# B&R Automation Studio project NAELD004C00R10L518F00 (part 4)

### Update LogProgram.txt
```
25/9/2023
Solved Inlet Shutter buffer empty close
added interlock to stop traverser and lifter when left or clear sensor sensed

2023-08-21, 2023-09-04, 2023-09-06   (R10)
DInput ,Doutput, OpsLifTrav - added outletshutter 2 (0276)
NtParam,UI - added Trolleylck 1&2 (0258)
UI,mcparam - added lane b fix to fix offset
UI - R to L
2023-09-04
UI - update 0258a topview position, teach picture
OpsMagConvLD1, LD2 - added p_bLinkTrolleyLckPrep
MtrPshr - MtrPshrActRet - added iRetSlwTor
Act_OptP0001Startup - Changed to AND gate.
2023-09-06
p0200 - added manual unlock trolley btn.

2023-07-31 (R9)
DInput - Act_Background - Start up buzzer update
UI - Act_Background - P1000_LangTime - Update the arrangement and display of the languagues and time
Ntparam - Add Chinese & German prep
AutoRcp - update structure , ntparam added eAutoRcpPrecededBy

2023_07_26 continue(R8) General_update
    > Update
            Manual accept for
            1) LFFollower,Follower1,Follower2,etc:Act_Background_AccData
            2) LCSLF:Act_Main
            3) USHermes: Act_Background_AccData

            HMI:
            1) Act_OptP0200ToP0201AccDat(Name based on Project)

2023-07-03 (R8)
-Auto Rcp (Compatiple only with Horizontal Hermes 1.3)
- Magazine auto Calculated width,min,max,pitch based on Board Available and Board Forecast
- Magazine Properties Retain Function
-SvyHermes Board Arrived,Board depart (Slotid,Magazaine ID)
-OPCUA AGV with RFID, read RFID tag when enter, write when exit
-Adding Magazine Exiting with buffer full,release magazine, AGV ready signal , product different (Auto Rcp)
- Error Handling for AutoRcp (Under Testing)
- Tuning MtrPshr
Commission line (_S0)
-MtrPshr - to solve alarm triggered when powered on
-Buffer1,2,3,4 - update Act_Initial diNxtUnloadSlt value.
-OpsTravLifLD - Rls button during readRFID
(_S1)
-Hermes<> smema transition to flush out magazine.
-Debug shutter close when puller extend
(_S2)
-Remove release btn mask.
-Resolved the last board with same width board available. (DSHermes)
(_S3)	2023-07-26
-AutoRcp - Act_Background2 -added p_diRequestedMinSlt when 5mm / 30mm btm clearance
-Debug the right sensor false triggered. (NOT(p_bConvHvBrd)) ,allowed reach ds position without active right sensor
(_S4) 2023-08-11
-Buffer 1,2,3 - Act_Background - added diCurrSltHermes
-DSHermes - seq - boardForcastID - No need sBoardID
			-ProcessData - added timer to reset bSendBFId (Forecast ID)
-SvyHermes - Act_Link - boardArrived - channge to p_bPullerRetRS
-OpsTravLifLD - TravLifLDStep1InletPneuCls - avoid keep open when no curtain sensor
-UI - update product name to WorkOrderId (in Hermes) (done B02,B03)

2023-06-05, 2023-06-14 (R7) --
NtParam - added hermes 1.3 supervisory
		- added shutter2,3 prep
		- added customerReq
AutoRcp - New package.

2023-05-17 (R6) -- .
-Debug the right sensor false triggered. (NOT(p_bConvHvBrd AND p_bRightSen))
OpsTravLifLD -- Added TravLifLDStep1DSSigRechk > TravLifLDStep1ConvEntBrdLostErr
Visu - Show the DBAOnRgt sensor in machine param.
OpsMagConvLD1,2,3 -Added downpulse for clampDetect sensor when magazine pre-exit
P0800, OpsMagConvLD1,2,3 - Updated set magEmpty at magInfo during run.
NtParam - Added eCustomerReq
OpsMagConvLD1 - Act_OpsInfo - Catered 2 empty magazine only buzzer. (BChina)
OpsTravLifLD -- added p_siCntrPullLmt and fbCTDPullLmt

2023-05-08 (R5) --
UI - Act_OptP0400Load.st - Avoid prompt LF message box when error.
OpsTravLifLD - Act_Link - Add a_bRlsMagBtn[1,2,3]
OpsMagConvLD1,2,3 - Act_OpsRun - Added condition on bRlsMagAllw.
HWInfo - Generate MacAddr file.

2023-3-22 (R4) --
Alarm
-Alarm.var added global variable to link text snippet alarm UI
-Act_Background - Recovery list changed to Alarm Error Code
-UI P0200 - change recovery text from string to text group
-UI P0600 - Trigger alarm using bAlm,bWarning,Errcode replacing the original string
-UI P0600 - Adding additional button to check alarm history
-UI Visu  - P0200,P0600 Using given Visu Alarm component instead of string text as the Alarm table

2023-03-15 (R4) --
OpsMagConvLD1,2,3,4 -- added p_bProjLifTravMnlLoad for non roller condition
CPU.sw -- PushPull Cycle time move up to 20 ms same as PullConv

2023-03-03 (R4) --
-UPDATE outstanding:
OpsMagConvLD1,2,3 - Act_OpsRun.st - Make unclamp top clamper when orientation / height sensor fail to sense.
									-LD2 ,3  -Rectified the height sensor alarm when condition not meet.
OpsTravLifLD - Act_OpsSubRun1.st - Catered unclamp(OpsMagConvLD1,2,3) when width check error.
Visu, P0900 , P0201 - Added magazine width check sensor IO.
P0202,P0203,P0204 - Rectified blank IO (Top Rmt Unclamp Sensor)
P1026 ,P1031 - Act_Main, Exit , FBCtrl - Add Bypass curtain sensor on all teaching pages.
DOutput - Act_Link - Allowed UI ctrl in stop mode.
OpsMagConvLD1,2,3 - Act_OpsRun.st - Add fbSelClmpTm wait for penumatic full clamp.
									- Make unclamp fix clamper when orientation / height sensor fail to sense.
PullConv - Local.var - Rearrange the offset text. (puller is Extending/ Retracting)

2023-02-23
LF 	- Act_InitGlobal	- Added p_eProdRcpStat, p_eProdRcpStatus, p_eLinkUIProdRcpAct, p_tyProdRcpCurrRcpWr
	- InputRef_Link		- Added ref variables based on declaration in Act_InitGlobal.
	- Act_Background_AccDat	- Re-adjusted usiProdAccDatStep, and additional usiProdAccDatStep for ProdRcpActWriteCurrRcpParam ProdRcp's Action

**Search Funciton Update** - NtRecipe 5.00.5 (L517)
- ProdRcp - Act_Main & Local.var
- Act_EntP1040Disp
- Act_OptP1040Save
- Act_OptP1040Del
- Act_OptP1040ToXML
- Act_OptP1040FromXML
- Act_EntP0400Disp
2023-01-17 (ANGSY)
UI - Act_Background - Act_OptP1080EditUsr - Add tyStringPw.sValue for every cases of tyP1080UsrMgmt.tyUsrMgmt.tyDrpDnLvl.usiValueIdx
										  - Uncomment tyP1080UsrMgmt.tyEdit.tyStringPw.sValue := '';
- Shift bDBAOnRgtSen from NtParam to McParam
- FTP drive migrate to F drive
--##

2022-12-07 (R3)
Ui - optimization(P0202 ,P0930,P0931, P0932),P0937 -update puller go width
NtParam - Added tyPPTorqParam
Pneu2SenInShutter2 - disabled when single inlet used.
Pneu2SenInShutter3 - disabled when single inlet used.
OpsTravLifLD - OpsRun - added MagPlat_Step1EntBrd, MagPlat_Step1InletPneuCls, MagPlat_Step1InletPneuOpn. (for magazine platform)

2022-09-24,2022-09-25,2022-10-12 (R2)
Trav - Rearrange the alarm list.
OpsTravLifLD - Integrate the individual shutter, cutain sensor feature. -Act_background
			 - Integrate magazine width check
MagConv2Clp1,2,3,4 - Reaccess the Clamping sensor.
PullerPusher - Act_Link - Include interrupt sensor with individual shutter.
			 - Act_RstErr - Reset diJogVel_60FF for recovery.
MagConv2Clp1,2,3 - MagConv2ClpActEntStopClp - changed to Fix clamp then remote clmap.
MagConv2Clp1,2,3 - MagConv2ClpActEntStopClp,MagConv2ClpActEntStopClp - add curtain interrupt for safety clamp
PullConv - Added ConvActInitPuller1 action.
Follower2 - Act_Link - Added p_bAccNewRcpCond.

2022-09-15 (R1)
Buffer 1;2;3;4 - Act_Main - BufferActUnload -make Slt to Slt as positive
Physical view - FTP server - added user for FTP access ProductRecipeXml

2022-03-24 (NAELD004-R0)
Act_Main_P0200 - added RS232Prep and WorkOrder string on barcodeScan
Act_OptP0200BarCodeChgRcp - added bWorkOrderDisp.
Added Act_OptP0200WorkOrderToLMC.st
PullConv - Hold postition when Antijam activated.

2022-03-14
ProdRcp - Act_Main, Local.var
MagRcp - Act_Main, Local.var

2022-02-17
LFFollower, Follower1 - Act_Background - Add p_bDBAOnWOAllign to fbFolllower to send DBA even width check sensor is not alligned.
CANOpenServo - Act_Background - Add error code for Estun Servo Motor.
				              - Reset control word 6040.4 to 0 when servo motor is in position

2021-09-30
Hermes Program - Update
USHermes Program - Update
DSHermes Program - Update
RmtHermes Program - Update
SvyHermes Program - *NEW*
NtParam  - Add new variables for Hermes v1.3
McParam  - Update
Alarm - Update
Startup - Update
UI HMI & Program P0201 - Update
UI HMI & Program P1021 - Update
UI HMI & Program P1022 - Update
UI HMI & Program P1023 - Update

2021-09-02
Revision - R15 , L512
- Width Offset move to NtParam
- Add BadBrdRedLight in NtParam and P0200 for 2021-0532G.
- McMode2 for 2021-0532G in P0201,P0400,P1021,P1040
LFLeader, LFFollower - Local,Input_Ref variables - Modify Product Recipe Related Variables to STRING[254]
LFFollower - Act_Background - Modify bUSAllow To Include p_bInternalReqProdRcpDiff

2021-08-31
Revision - R14 , L512
LFFollower - Update Act_Background
Follower1 - Update Act_Background
- Update NtUSB to 5.00.5
- Update NtLF to 5.01.4
- OPC-UA Security Policy Basic256 Sha256 prohibited

2021-08-02
USB scanner function added.
AIV OPCUA, Hardwired IO and Disabled function added.
IO assignment at physical view changes without alter the value of digital input and digital output at NtParam.

2021-04-06
UI - Visu - Update for 254 Prod Rcp Pop Up
UI - Act_Background - ADD Act_OptP0400RcpPopUp.st & Act_OptP1040RcpPopUp.st & Update Act_OptP0400Preview.st for 254 Prod Rcp Pop Up

2021-02-24
LFLeader - Act_Main - add input to select sequential mode (one time or always active)

2021-02-17
CANOpenServo - Act_Background - PosDiff updated from 50 to 500.
			 - Act_Alarm - udiCode change to 10299
			 - Local.var - update alarm message a_tyAlmText[10298] and a_tyAlmText[10299]

2020-12-14
Update in Act_ChgPage & Act_OptP00001Startup

2020-11-11
Tuning.diAsdaA2FirstTorqueCmd default setting is 300 in NtParam for all Delta servo motor.

2020-10-05
Startup - Act_Main_GetHWInfo - Debug Steps In Network Recovering
LFLeader - Act_Initial, Act_Background_Process and Local.var - Rename and change the type of fbBlkUS to fbBlkUSDS
LFFollower, Follower1 - Act_Background, Act_Background_AccData - Add bLeaderOnline replacing the direct usage of tyLeaderInfo.bOnline
TLBuz - Add Buzzer For All Act_Backgrounds Change Manual Mode Towerlight To Cater For Error Indication
HWInfo - Act_Main - Add IF-ELSE Statement For Simulation, Update Alarm Code for fbGetETHConfigMode & fbSetETHConfigMode
		 Local.var - Add New Alarm Code fbGetETHConfigMode & fbSetETHConfigMode

2020-09-22
LFFollower - Reset bLeaderSeqCtrlInActive in Act_Main_Disable.
HWInfo.typ - Add One Enumeration (eNetworkConfigMod) & Two Actions (fbGetETHConfigMode and fbSetETHConfigMode) - Retrieve Or Set Network Configuration Of The PLC.
HWInfo Init, InitGlobal, InitLocal, Act Main, Act_Initial, Local.var and InputRef.var - Add The Additional Actions Related Variables
McParam  - McParam.typ Add eNetworkMod in tyMcParam.
NtParam  - NtParam.typ Add tyNetworkMOde (UILmt) in tyNtParam.
Startup	   - InitGlobal, InitLocal, Act_Main_GetHWInfo - Add Function To Load Saved Network Configuration s When New Configuration Detected.
		   InputRef_Link.var, InputRef.var & Local.var - Add New Startup Function Variables.

2020-09-16
McParam  - McParam.typ Add sIPAddr & sSubnetMask in tyMcParam.
Startup	 - Init, InitGlobal, InitLocal, Act_Main_GetHWInfo - Add Function To Load Saved IP Parameters When New IP Detected.
		   InputRef_Link.var, InputRef.var & Local.var - Add New HWInfo Function Variables.

2020-09-10
USHermes - Init, Cyclic, Act_Background_TCPConnect, Act_Alarm5 - Improvise Alarm For Connection Lost.
		   Local.var - Add New Alarm Variables & Modify Alarm Text.
DSHermes - Init, Cyclic, Act_Background_TCPListen, Act_Alarm4 - Improvise Alarm For Connection Lost.
		   Local.var - Add New Alarm Variables & Modify Alarm Text.

2020-08-17
LibVer - Act_Main - Modify Function To Function Block In LibVerActReadChk.
		 Act_Initial - Initialize Newly Added Function Blocks.
		 Local.var - Declare New Function Blocks.

2020-08-06
NtParam.typ - Add Two Actions (NtParamSave and NtParamLoad) - Export and import NtParam in XML Format
NtParam Act Main, Act_Initial, tyNtParam, InitLocal, Local.var and InputRef.var - Add The Additional Actions Related Variables
TLBuz - All Act_Backgrounds Change Manual Mode Towerlight To Cater For Error Indication
LFLeader - Add More Tags For Improving Leader Follower Concept, Modify p_diReqProdWidth To Use Downstream Width
LFFollower, Follower 1 	- Add fbOnlineChk For Leader Online Status
						- Modify Act_Initial,Act_Background, Act_Background_AccData
						- Add eCurrMachineStat For Status Indication
ProdRcp.typ		- Add second width
LibVer - Act_Main - Modify LibVerActReadChk, Add Step To Check File Validity.
		 Local.var - Add Alarm Text For File Coruption.

2020-07-24
MagRcp -  Add One Action in Act Main - MagRcpActSort
ProdRcp, MagRcp - p_sSearch and sSearch in Local changed to STRING[254]
ProdRcp, MagRcp - sRcpNm for RcpParam in both ProdRcp.typ and MagRcp.typ temporary changed to STRING[30]

2020-06-30
Revert Traverser Main.st and AWClose Background.st program.
Add Estun error code "65362: sAxisErrTxt := 'Torque output alarm'";

2020-06-08
ProdRcp - Increase Product Recipe Name Length to 254, Add Two Actions in Act Main - ProdRcpActSort & ProdRcpActEndCharFilter
LibVer - Act_Main - LibVerActReadChk, made error if library data files corrupted.

2020-06-05
MagConv - Update the Status of Mag Conv.Add one Action - MagConvActEntToMid.

2020-06-01
Stepper - New package for stepper control.
MotorBrk - Renewed package. Added MotorBrkActSetMtrDirOrCCW1 and MotorBrkActRstMtrDirOrCCW1.
	 	 - Modified fbRotCW and fbRotCCW and the access type to fbConvSenToSenBrkTm2Lmt.
	 	 - Added diMtrSigOnDlyTm (500), diMtrDirOffDlyTm (500), diMtrBrkOnDlyTm(100).

2020-04-28
MagConv - Add MagConvActEntToMid Action.

2020-03-20
NtParam  - Add the selection of Motor model.

2020-03-16
TLBuz - Add two inputs for buzzer behaviour, towerlight flash function to act_background and reset fbwarning.

2019-12-24
LFLeader - Remove fbBlkDS2 in Act_Initial & Act_Background_Process, add pa_bLFOnline in Act_Background_Process

2019-10-31
TLBuz - Regroup Structure Into Nutek, Aptiv & MEK.
MagConv - Separate Program Into MagConv1Clamper & MagConv2Clamper.

2019-10-21
MagConv - Improve with Action MagConvActPreExit & MagConvActPreExitClpr.
LFFollower - Improve Change All Function Without Manually Accept Data.
LFLeader - Add Second Oven Index, Improve Change All Function Without Manually Accept Data.
OpcUaMap.uad - Enable bBypassMnlAccDat Tag Name.
Startup - Act_Main_SDOWrite, Remove SDOWrite.
CANOpenServo - Change Structure Of SDOWrite And Abnormal Movement.

2019-07-30
CANOpenServo - Due To Upgrade of NtMotion.

2019-07-18
LFFollower - Act_Link, Minor debug.

2019-07-15
LCS - Act_Link, Check Recipe Name Must Not Exceed 15 Char.

2019-07-10
LCS - Add More Parameter For Live Data.

2019-07-04
LFFollower - Improve of Recipe Compare Method For p_tyInternalReqProdRcp, tyUpdtProdRcp & tyRlsBrdProdRcpNm.

2019-07-03
LFFollower - Improve Act_Background To Check Whole Product Recipe Different Instead of Name & Width Only.
Buffer - Add p_tyBufferStat & p_tyDispBuffer And Improve For Two Program Control One Memory.

2019-06-28
USHermes - Improve of Act_Background_AccData.
DSHermes - Move of Act_Background_ChgConfig.
Buffer - Improve of bParamDiff Condition.
LCSLF - Improve of LCSActRunProd.

2019-06-27
LFFollower - Improvement To Change Name & Width To Whole Product Recipe Type.

2019-06-17
Conv - Add Two Action : ConvActEntToInOff & ConvActRevImmedStart.

2019-06-12
LFFollower - Add Act_Background_ChkRlsBrd. Improvement of Act_Background_UpdtData.
LCSLF - Add Update Data in Act_Background.

2019-06-11
TLBuz - Modify ChgRcp.
LFFollower - Improvement of UpdtData.

2019-06-10
ProdRcp - Update tyCurrRcp To a_tyCurrRcp (Array).
LFFollower - Add p_bInternalUse.
USHermes - Add p_bInternalUse.
DSHermes - Add p_bInternalUse.

2019-06-07
TLBuz - Add Warning & ChgRcp.
TCP - Add Start Code & End Code Checking.
Buffer - Improve bParamDiff. Add bFIFOOld.

2019-06-04
USHermes - Improvement At Accept Date (Act_Background_AccData).

2019-06-02
TCP - New.

2019-05-30
Hermes - Debug CheckAlive. SequenceTO Start Only After Connection Establish.
Flatstream - Debug Act_Main.
USHermes - Update Act_Link to Accept New Recipe.

2019-05-29
DVFrame - Change From RS232. Improvement & Debug.
Flatstream - New.

2019-05-28
MagConv - Add MagConvActInitClpStop.
DCConv - Improvement of DC Motor Alarm Trigger Time.
LFFollower - Improve of Act_Background.
LCS - Add "Warning" & "Info" For Live Data.

2019-05-27
LFFollower - Debug Act_Link.
LCS - Debug Act_Link. Add sErrMsg.
Buffer - Debug Act_Main_Bffr. Add bMagRemoved.
Data - Update of Default User.dat.

2019-05-24
LFFollower - Improve of Act_Background.
MagConv - Add MagConvActEntClpStop.
TLBuz - Modify Warning Condition.

2019-05-22
OpcUaMap.uad - Update Tag Name.
LF - Modify Set Time. Improve Of Act_Background for Accept Data.
LFLeader - Add New Tag Name.
Time - Update of Act_InitGlobal For LF Sync Time.
LCS - Update To Reset If Receive Idle From LCS.

2019-05-21
RS232 - Add FullReadUntilValid.
LCS - Move Some Program From Act_Background To Act_Link. Bug Fixed.

2019-05-20
RS232 - Modify to work with start code & end code.
ProdRcp - Modify on dtLastModified in Act_LinkAction.
LCS - Act_Background Show Boolean & dtLastModified Working Sample. Add Function Enable.
TLBuz - Add Aptiv Mode.

2019-05-18
Buffer - Check Next Unload Ignore Product Name.

2019-05-15
OvenInfo - Improve of Act_Background.
Buffer - Add bParamDiff to check current parameter and request parameter different.

2019-05-14
LCS - Update Act_InitGlobal.
RS232 - New.

2019-05-11
LFFollower - Improve And Able To Ignore MagRcp If Necessary.

2019-05-10
TLBuz - Add Simulation Mode.
ProdRcp - Improve Act_LinkAction.
Buffer - Improve Act_LinkAction.
HWInfo - Improve Act_Main While In Simulation.

2019-05-09
CANOpenServo - Improve of Error Axis Move Abnormally By External Force (10000).
ProdRcp - Debug Write Recipe. Add Save List.
MagRcp - Debug Write Recipe. Add Save List.
UsrFolder - Create LCS Directory.
Startup - Act_Main_UsrFolder, Create LCS Directory.
Alarm - Combine Two Alarm Info.

2019-05-08
RmtHermes - Debug Log title.
UsrMgmt - Add Access Right Output.

2019-05-07
MagConv - Debug.
ConvBffr - Add Individual Have Board Output.
LF - Major update.
LCSLF - Change Name to tyCurrProdRcp.
ProdRcp - Add Write Recipe Parameter.
MagRcp - Add Write Recipe Parameter.
LCS - Update to match LCS (PC).

2019-05-04
MagRcp - Split Current Magazine Recipe From McParam.
ProdRcp - Split Current Product Recipe From McParam.
UsrMgmt - Split Access Right From McParam. Remove Nutek User.
Hermes - Split Configuration From McParam. Add RmtHermes.
Startup - Split Parameters From McParam. Add RmtHermes.
Remove "File Device" "NutekUser". Please Refer Configuration "4PPC30_043F_21F001".

2019-05-01
Hermes - Log file change to day instead of hour. Due to startup too long to check old log when production run for long.

2019-04-30
LCS - Improve To Match LCS (PC).
LFLeader - Make a_tyFollowerToLeaderTag as Output.
All - sStatTxt & a_sStatText Change To String[200].
ProdRcp - Modify For LCS.

2019-04-28
MpProdRcp - New.
Add "Config.mprecipexml" Under Configuration View > mapp. Please Refer Configuration "4PPC30_043F_21F001".
Add "File devices" For "MpProdRcp". Please Refer Configuration "4PPC30_043F_21F001".
Startup - Modify Due To MpProdRcp.

2019-04-27
DSSMEMA - Update due to NtSMEMA upgrade.

2019-04-26
Buffer - Debug tyBuffer to p_tyBuffer. Improve bLastProductUnload Condition In Unload Board.
Startup - Get Retain ConvBffr.
ConvBffr - Update Link with Startup. Improve bLastProduct Condition In Remove Board. Add Have Board Output.
LFFollower - Improve Act_LinkEn. Add Condition in Act_Link to update current recipe into leader tag.

2019-04-25
LibVer - Modify To Move LibVer From "Private" To "User".
Update "File devices" For "LibVer". Please Refer Configuration "4PPC30_043F_21F001".
Add "File devices" For "LCS". Please Refer Configuration "4PPC30_043F_21F001".
Modify "FTP Server" "Users". Please Refer Configuration "4PPC30_043F_21F001".
Modify "OpcUaMap.uad". Please Refer Configuration "4PPC30_043F_21F001".
LFLeader - Improvement.

2019-04-24
CANOpenServo - Add actual limit sensor output.
ProdRcp - Add "Add" & "Edit" action. Improve of Act_LinkAction to suit LCS.
LCS - New.

2019-04-23
LFLeader - New.

2019-04-21
USHermes - Modify Alarm Info.
LFFollower - New.

2019-04-18
ConvBffr - New.
Buffer - Change of NtBffr.

2019-04-17
CANOpenServo - Remove Extra Homing Parameter, All Use Under tyMotionCANParamInHm.

2019-04-16
Operations - Remove Accept Data & New Data.
Hermes - Debug Log File. Modify Accept Data.

2019-04-11
USHermes - Debug Log by adding step. Add p_bAccDataRdy.
DSHermes - Debug Log by adding step.

2019-04-10
Startup - bNtSettingsLoadDone should be FALSE as default.

2019-04-09
Ops2 - Update of p_bAccDat interlock by Ops1.
USHermes - Update AccDatStep in Act_Link. Remove p_bChkBrdAvl. eStatus2 = Error then bRdyRcv = false. Update Act_Background_BoardAvailableChk. Add Manual Accept Data.
DSHermes - Make local.var BoardAvailable new board parameter to default value.
NtParam - Change of Act_LinkAction.
TLBuz - Change of Act_LinkAction.
Buffer - Change of Act_LinkAction.
Conv - Change of Act_LinkAction.
DCConv - Change of Act_LinkAction.
MagConv - Change of Act_LinkAction.
MotorBrk - Change of Act_LinkAction.
ConvSpd - Change of Act_LinkAction.
SMEMA - Change of Act_LinkAction.
Pneu - Change of Act_LinkAction.
CANOpenServo - Change of Act_LinkAction.
Hermes - Change of Act_LinkAction.

2019-04-08
DSHermes - Minor debug on fbParseBrdAvlExternal.
Hermes - Add program Hermes for board available memory use.
Startup - Due to change of Hermes.

2019-04-04
OvenInfo - Add p_bBGRun.
Startup - Change eStartupStep member order for better display in UI.
UsrMgmt - Add UsrMgmtActUsrBypassLogin & UsrMgmtActNtBypassLogin.
DSHermes - Debug BoardAvailable for "New" and "External".
UI - Remove Not Use Page.

2019-03-29
All - Add Act_LinkAction.

2019-03-28
Startup - Change "DelOldLogFile" to "Alarm". Add "Hermes". Error will reset Action to IDLE.

2019-03-25
All - Change Action become input. Merge Alarm Text & Recovery Text into one type.

2019-03-22
Startup - Add bNtSettingsLoadDone. Move StartupStepParameter after StartupStepUsrFolder in Act_Main.st.
All - Update to match latest method of NtParam.

2019-03-16
Startup - Act_Main_Bffr. Add BufferActBGStartCoolFan in Step 8.

2019-03-15
Hermes - New Release

2019-03-13
UsrFolder - Debug of Log directory path. Add "FileDevice" for "Log".

2019-03-11
DCConv - Minor debug.

2019-02-26
AWClose - Minor debug.

2019-02-23
Alarm - Minor debug.
UsrFolder - Add Create Log Directory.
Startup - Improve of "Act_Main_UsrFolder" due to UsrFolder update.

2019-02-22
CANOpenServo - Change of Act_Action.

2019-02-21
DOutput - Add Act_Link.

2019-02-20
DCConv - Debug of ConvEngage.
CANOpenServo - fbModuleOK delay time change to 5s.

2019-02-19
CANOpenServo - Reset Error need to reset control word 6040.
TLBuz - Improve of condition while p_bManual = True.

2019-02-18
Buffer - Add background control of cool fan run.

2019-02-15
Conv - Improve of condition while p_bManual = True.
DCConv - Improve of condition while p_bManual = True.
MagConv - Improve of condition while p_bManual = True.
MotorBrk - Improve of condition while p_bManual = True.
SMEMA - Improve of condition while p_bManual = True.

2019-02-14
ConvSpd - Improve of condition while p_bManual = TRUE.
Change of Cyclic Time.
CANOpenServo - Change of Position Different Threshold.
Convert Library Into Binary

2019-02-11
TLBuz - Warning Rest Time Change To 5s.
Buffer - Add Magazine Present Timer.

2019-01-27
Buffer - Add error code.

2019-01-26
Buffer - Debug.

2019-01-25
Buffer - Debug a_bSkip array size.
Lifter - Debug Act_Background.
User.dat & NtUser.dat update.

2019-01-24
Pneu - Modify Cyclic for disable.
AW - Add GoWidthOff to turn off motor after auto width move.
Lifter - Debug.
Traverser - Debug.
Buffer - Debug. Add background update display.
OvenInfo - Modify Act_Main_Disable.

2019-01-23
Lifter - Major debug in slot calculation. Add FullMovRel.
CANOpenServo - Debug reset error. Debug Act_Alarm.
DCConv - Debug reset error.
Machine - Debug reset error.
Operation - Debug reset error.

2019-01-22
CANOpenServo - Minor debug.

2019-01-21
DInput - Debug reset error.
CANOpenServo - Add eMainStatus. Add bJogging.
Time - Add eMainStatus.
Operations - Rename eStatus & udiStatus.

2019-01-20
Operations - Update Structure.
SMEMA - Update due to Library update.
Buffer - Add error code.

2019-01-19
TLBuz - Add Warning.

2019-01-18
RstErr - Act_Main update.
CANOpenServo - Add output. Set Default Value for siModOfOptDisp_6061:=6.
Change of Cyclic time.
Buffer - Update Local.var
Add file for NtUser, LibrariesVersion & User.
Conv - Add Pneu status output.
DCConv - Add Pneu status output.
Operations - Modify structure in Cyclic.

2019-01-17
DCConv - Act_Main debug.

2019-01-16
Trav - Remove diPitch.
Lifter - Remove diPitch.
Operations - Modify Reset methos.

2019-01-15
McParam - File name as input.
NtParam - File name as input.
Buffer - File name as input.
Operations - Add bAccData.

2019-01-14
Operations - Update Alarm & Sequence.
SMEMA - bTimer & bVirtual as output. Debug Act_Background timer interlock.

2019-01-12
Conv - Convert time out type.
DCConv - Convert time out type.
MagConv - Convert time out type.
OvenInfo - diBrdInOven change to retain.
SMEMA - Update timer condition. Add bComplSigOn.
Startup - Debug for HWInfo.

2019-01-11
SMEMA - Minor debug. Add Act_LinkEn.
Operations - Add alarm. Add Act_LinkEn.
MagRcp - Add Act_LinkEn.
OvenInfo - Add Act_LinkEn. Minor debug.
Conv - Add Act_LinkEn. Add conveyor time out.
DCConv - Add Act_LinkEn. Add conveyor time out.
MagConv - Add Act_LinkEn. Add conveyor time out.
MotorBrk - Add Act_LinkEn.
ConvSpd - Add Act_LinkEn.
RS232Mirtec - Add Act_LinkEn.
Pneu - Add Act_LinkEn.
CANOpenServo - Add Act_LinkEn. Major Update.

2019-01-10
McParam - Remove ProdRcpWrite & MagRcpWrite.
OvenInfo - Act_Main modify for change of eStat.
Conv - Act_Main modify for change of eStat.
DCConv - Act_Main modify for change of eStat.
MagConv - Act_Main modify for change of eStat.
MotorBrk - Act_Main modify for change of eStat.
ConvSpd - Act_Main modify for change of eStat.
SMEMA - Act_Main modify for change of eStat.
DOutput - Act_Main modify for change of eStat.
Pneu - Act_Main modify for change of eStat.
Operations - Act_Main modify for change of eStat.

2019-01-09
AW - Update bWidthPosDiff when disable.
Lifter - Update bSltPosDiff when disable.
Conv - Add bGdBrdInit. Debug tMtrOffDlyTm. Improve Act_Action to let eStatus = DONE also able change eStat directly.
DCConv - Add bGdBrdInit. Improve Act_Action to let eStatus = DONE also able change eStat directly.
SMEMA - Add tRstDlyTm. Improve Act_Action to let eStatus = DONE also able change eStat directly.
Operations - Add Act_Main_Disable. Improve Act_Action to let eStatus = DONE also able change eStat directly.
TLBuz - Improve Act_Action to let eStatus = DONE also able change eStat directly.
OvenInfo - Improve Act_Action to let eStatus = DONE also able change eStat directly.
MagConv - Improve Act_Action to let eStatus = DONE also able change eStat directly.
MotorBrk - Improve Act_Action to let eStatus = DONE also able change eStat directly.
ConvSpd - Improve Act_Action to let eStatus = DONE also able change eStat directly.
DOutput - Improve Act_Action to let eStatus = DONE also able change eStat directly.
Pneu - Improve Act_Action to let eStatus = DONE also able change eStat directly.

2019-01-08 //Until Here////
DOutput - Add output.
SMEMA - bTimer will be trigger only during SMEMAActRun.
Operations - Combine Ops1 & Ops2 into Ops.

2019-01-07
SMEMA - Add bUSRdy, bUSGdBrdRdy & bDSRdy for USSMEMA & DSSMEMA.
Conv - Add tMtrOffDlyTm.
DCConv - Add tMtrOffDlyTm.
MagConv - Add tMtrOffDlyTm.
Time - Combine Error
CANOpenServo - Combine Error
Alarm - Remove link data.

2019-01-04
Machine - Debug Act_Alarm1.
Time - Debug Init.st.
Operations - Debug Ops1 > Act_Main. Add sStepTxt into Act_Main. Add Act_Dummy.
Conv - Due to NtConv update, add one more type of Exit.
DCConv - Due to NtConv update, add one more type of Exit.
MagConv - Due to NtConv update, add one more type of Exit.
SMEMA - Add Timer & Virtual.

2019-01-03
Machine - Debug Act_Alarm & Act_Alarm1. Modify background error handling.
CANOpenServo - Modify background error handling. Update sStatTxt in Act_Initial.
AW - Replace diStandPitchInUM (Input) to diPitchInUM (Local).
Time - Modify background error handling. Update sStatTxt in Act_Initial.
DCConv - Modify background error handling. Update sStatTxt in Act_Initial.
DInput - Modify background error handling.
UsrMgmt - Update sStatTxt in Act_Initial.
McParam - Update sStatTxt in Act_Initial.
NtParam - Update sStatTxt in Act_Initial.
ProdRcp - Update sStatTxt in Act_Initial.
MagRcp - Update sStatTxt in Act_Initial.
HWInfo - Update sStatTxt in Act_Initial.
UsrFolder - Update sStatTxt in Act_Initial.
LibVer - Update sStatTxt in Act_Initial.
General - Update sStatTxt in Act_Initial.
TLBuz - Update sStatTxt in Act_Initial.
OvenInfo - Update sStatTxt in Act_Initial.
Buffer - Update sStatTxt in Act_Initial.
RstErr - Update sStatTxt in Act_Initial.
Conv - Update sStatTxt in Act_Initial.
MagConv - Update sStatTxt in Act_Initial.
MotorBrk - Update sStatTxt in Act_Initial.
ConvSpd - Update sStatTxt in Act_Initial.
Alarm - Update sStatTxt in Act_Initial.
RS232Mirtec - Update sStatTxt in Act_Initial.
SMEMA - Update sStatTxt in Act_Initial.
UI - Update sStatTxt in Act_Initial.
DOutput - Update sStatTxt in Act_Initial.
Pneu - Update sStatTxt in Act_Initial.
Operations - Update sStatTxt in Act_Initial.
Startup - Update sStatTxt in Act_Initial.

2019-01-02
UsrMgmt - Change of sStatTxt update.
McParam - Change of sStatTxt update.
NtParam - Change of sStatTxt update.
ProdRcp - Change of sStatTxt update.
MagRcp - Change of sStatTxt update.
Time - Change of sStatTxt update.
HWInfo - Change of sStatTxt update.
UsrFolder - Change of sStatTxt update.
LibVer - Change of sStatTxt update.
General - Change of sStatTxt update.
TLBuz - Change of sStatTxt update.
OvenInfo - Change of sStatTxt update.
Buffer - Change of sStatTxt update.
RstErr - Change of sStatTxt update.
Conv - Change of sStatTxt update.
DCConv - Change of sStatTxt update.
MagConv - Change of sStatTxt update.
MotorBrk - Change of sStatTxt update.
ConvSpd - Change of sStatTxt update.
Alarm - Change of sStatTxt update.
RS232Mirtec - Change of sStatTxt update.
SMEMA - Change of sStatTxt update.
UI - Change of sStatTxt update.
DOutput - Change of sStatTxt update.
Pneu - Change of sStatTxt update.
Operations - Change of sStatTxt update.
CANOpenServo - Change of sStatTxt update. Update eStatus to Busy while running.
Startup - Change of sStatTxt update.

2018-12-31
CANOpenServo - Seperate input reference.

2018-12-27
Time - Remove bBGRun.
TLBuz - Remove bBGRun. Add manual reset.
OvenInfo - Background direct link to input bPrepExtdd, bEnExtdd & bDisExtdd. Add manual reset.
Buffer - Background Cool Fan Control direct link to input bPrepCoolTm & bCoolFanTm.
DCConv - Remove bBGRun. Add manual reset.
AlarmLog - Background run is control by Action.
Machine - Remove bBGRun.
SMEMA - Remove bBGRun. Add manual reset.
DInput - Remove bBGRun.
DOutput - Remove bBGRun. Add manual reset.
CANOpenServo - Remove bBGRun. Background run is control by Action. Add manual reset.
AW - Add bWidthPosDiff.
Lifter - Add bSltPosDiff.
Startup - Background run is control by Action. Shorten local variable name.
McParam - Add McParam program without Magazine (McParam2).
RstErr - Add manual reset.
Conv - Add manual reset.
MagConv - Add manual reset.
MotorBrk - Add manual reset.
ConvSpd - Add manual reset.
Pneu - Add manual reset.

2018-12-26
CPU - Update distribute of program in CPU. Update cyclic time.
FTP - Update of FTP server configurations.
Startup - Remove bStartupErr.
HWInfo - After set new IPAddr & Subnetmask will update output.
TLBuz - Rising of bManual will set Amber Light ON.
Conv - Remove functions reset in individual eStat.
MagConv - Remove functions reset in individual eStat.
MotorBrk - Remove functions reset in individual eStat.
DCConv - New program.
Operations - Update of OperationsActStep.

2018-12-24
Operations - Add bRun.Sequence will execute base on bRun instead of bStatusRun.

2018-12-21
Buffer - Add individual cooling fan control.
McParam - Move Hermes parameter to Hermes program type.
MagConv - Add bClprTwoOutputControl. Remove bClprUnclampCtrl.

2018-12-20
TLBuz - Add bMuteBuz.
OvenInfo - Add bDis.
Conv - Add bEn.
MagConv - Add bEn.
MotorBrk - Add bEn.
ConvSpd - Add bEn.
RS232Mirtec - Add bEn.
SMEMA - Add bDis.
Pneu - Add bEn.
CANOpenServo - Add bEn.
CANOpenServo - AutoWidth - Add diMaxWidthInUM, diMinWidthInUM, diWidthOffsetInUM & diStdPitch.
Operations - Add bPrep, bEn & bDis. Add OperationsStatusCycleStopping. Default Status is OperationsStatusStop. Add Boolean output for Status.
MagRcp - Change sDisplayInfo & Magazine Parameter.
Startup - Add bRun.

2018-12-14
RstErr - Add bManual to control reset of output in Idle. Reset output in Idle after ManualMode off.
Conv - Add bManual to control reset of output in Idle. Rename eAction. Reset output in Idle after ManualMode off.
ConvSpd - Add bManual to control reset of output in Idle. Reset output in Idle after ManualMode off.
MtrBrk - Add bManual to control reset of output in Idle. Rename eAction. Reset output in Idle after ManualMode off. Reset after change eStat.
MagConv - Add bManual to control reset of output in Idle. Rename eAction. Reset output in Idle after ManualMode off. Reset after change eStat.
OvenInfo - Set bOvenAllow to TRUE, if all functions not activated.
SMEMA - Reset output in Idle after ManualMode off.
Pneu - Add Extended & Retracted output.

2018-12-13
Conv - Change of Conv2Sen to Conv. Add Reject & Inspection functions. Add individual output control.
Pneu - Add bTwoCtrlIn & bTwoCtrlOut.
TLBuz - Add individual output control.
ConvSpd - Add individual output control.
OvenInfo - Add individual output control. Move functions into Act_Background.
RstErr - Add individual output control.
MtrBrk - Add individual output control.
MagConv - Add individual output control.
DOutput - Add individual output control.
SMEMA - Add individual output control.

2018-12-12
Startup - Add Logout during User Management Startup.
Time - Move Act_Background above Act_Main.
Buffer - Move Act_Background above Act_Main.
Alarm - Move Act_Background above Act_Main.
CANOpenServo - Move Act_Background above Act_Main.
Operations - Change of Conv2Sen to Conv.

2018-12-11
DOutput - Split to Act_InitGlobal & Act_InitLocal.
Pneu - Change in all program. Add Pneu3Sen program.
Operations - Update sample to 2 operations. Rename variable.
CANOpenServo - Rename variable.
```

- LibrariesVersion.dat (binary file, 2222 bytes)
### SoftwareVersion.var
```iecst
VAR CONSTANT
	sSWVersion : STRING[30] := 'NAELD004C00R10L518F00'; (*LifterPlatform and TraverseLifting*)
END_VAR
```

- Visualisation Logical/UI/Visu (not shown)

### UI.typ - Do Not Change!!!
```iecst
(*2019-03-25*)
(**)

TYPE
	eUIAction :
		(
		UIActIdle,
		UIActInitial
		);
END_TYPE

(**)
(*Data*)

TYPE
	eUIInitial :
		(
		UIInitialC0005,
		UIInitialC0007,
		UIInitialP0000,
		UIInitialP0002,
		UIInitialP0200,
		UIInitialP0201,
		UIInitialP0202,
		UIInitialP0203,
		UIInitialP0204,
		UIInitialP0205,
		UIInitialP0206,
		UIInitialP0300,
		UIInitialP0400,
		UIInitialP0410,
		UIInitialP0800,
		UIInitialP0900,
		UIInitialP0910,
		UIInitialP0920,
		UIInitialP0921,
		UIInitialP0923,
		UIInitialP0930,
		UIInitialP0931,
		UIInitialP0932,
		UIInitialP0933,
		UIInitialP0934,
		UIInitialP0935,
		UIInitialP0936,
		UIInitialP0937,
		UIInitialP0939,
		UIInitialP0940,
		UIInitialP0950,
		UIInitialP1000,
		UIInitialP1020,
		UIInitialP1021,
		UIInitialP1022,
		UIInitialP1023,
		UIInitialP1024,
		UIInitialP1025,
		UIInitialP1026,
		UIInitialP1027,
		UIInitialP1028,
		UIInitialP1030,
		UIInitialP1031,
		UIInitialP1040,
		UIInitialP1050,
		UIInitialP1080,
		UIInitialP1081,
		UIInitialDone
		);
END_TYPE

(*Global Alarm*)

TYPE
	tyUIAllAlm : 	STRUCT
		bAlm : ARRAY[0..9999]OF BOOL;
		bWarning : ARRAY[0..9999]OF BOOL;
	END_STRUCT;
END_TYPE
```

### UI.var - Change By Project
```iecst
(*2019-03-25*)
(**)
(*Action & State & Status*)
VAR
	p_UIStat : UDINT;
	p_UIStatus : UDINT;
	p_UIStatTxt : UDINT;
END_VAR
(**)
(*Alarm*)
(**)
(*Output*)
VAR
	p_UIStartupAct : UDINT;
	p_UISimuAct : UDINT;
	p_UIHWInfoAct : UDINT;
	p_UITLBuzAct : UDINT;
	p_UIRstErrAct : UDINT;
	p_UIProdRcpAct : UDINT;
	p_UIMpProdRcpAct : UDINT;
	p_UIMagRcpAct1 : UDINT;
	p_UIMagRcpAct : UDINT;
	p_UIMcParamAct : UDINT;
	p_UIUsrMgmtAct : UDINT;
	p_UIBuffer1Act : UDINT;
	p_UIBuffer2Act : UDINT;
	p_UIBuffer3Act : UDINT;
	p_UIBuffer4Act : UDINT;
	p_UIDSSMEMAAAct : UDINT;
	p_UIDSSMEMABAct : UDINT;
	p_UIInShutterAct : UDINT;
	p_UIInShutterAct2 : UDINT;
	p_UIInShutterAct3 : UDINT;
	p_UIOutShutterAct : UDINT;
	p_UIOutShutterAct2 : UDINT;
	p_UIPullerAct : UDINT;
	p_UIPullConvAct : UDINT;
	p_UIMagConvSelClp1Act : UDINT;
	p_UIMagConvSelClp2Act : UDINT;
	p_UIMagConvSelClp3Act : UDINT;
	p_UIMagConvSelClp4Act : UDINT;
	p_UIMagConv2Clp1Act : UDINT;
	p_UIMagConv2Clp2Act : UDINT;
	p_UIMagConv2Clp3Act : UDINT;
	p_UIMagConv2Clp4Act : UDINT;
	p_UIAWPushOrPullerAct : UDINT;
	p_UIAWOpenAct : UDINT;
	p_UILifterBtmAct : UDINT;
	p_UITravAct : UDINT;
	p_UIDOAct : UDINT;
	p_UIHermesAct : UDINT;
	p_UILFLeaderAct : UDINT;
	p_UIOpsAct : UDINT;
	p_UIFrmAct : UDINT;
	p_UIMtrPshrAct : UDINT;
	p_UIServoPPAct : UDINT;
END_VAR
(**)
VAR
	p_UIMnlMtrPshrRetSpd : UDINT;
	p_UIMnlMtrPshrRetTorq : UDINT;
END_VAR
(**)
VAR
	p_UIMcParamWr : UDINT;
	p_UINtWr : UDINT;
END_VAR
(**)
VAR
	p_UIProdRcpInfoIn : UDINT;
	p_UIProdRcpSearch : UDINT;
	p_UIProdRcpScan : UDINT;
	p_UIProdRcpCurrRcpWr : UDINT;
END_VAR
(**)
VAR
	p_UIMagRcpInfoIn : UDINT;
	p_UIMagRcpSearch : UDINT;
	p_UIMagRcpCurrRcpWr : UDINT;
END_VAR
(**)
VAR
	p_UIMagRcpInfoIn1 : UDINT;
	p_UIMagRcpSearch1 : UDINT;
	p_UIMagRcpCurrRcpWr1 : UDINT;
END_VAR
(**)
VAR
	p_UIUsrMgmtInfoIn : UDINT;
	p_UIUsrMgmtAccessRightLvl1Wr : UDINT;
	p_UIUsrMgmtAccessRightLvl2Wr : UDINT;
	p_UIUsrMgmtAccessRightLvl3Wr : UDINT;
END_VAR
(**)
VAR
	p_UIHermesDSParamWr : UDINT;
	p_UIHermesSvyParamWr : UDINT;
END_VAR
(**)
VAR
	P_UISectionLdr : UDINT;
END_VAR
(**)
VAR
	p_UISetIPAddr : UDINT;
	p_UISetSubnetMask : UDINT;
	p_UINetworkMode : UDINT;
END_VAR
(**)
VAR
	p_UIMnlMod : UDINT;
	p_UIUIMnlMod : UDINT;
	p_UIMuteBuz : UDINT;
	p_UISimuMod : UDINT;
END_VAR
(**)
VAR
	p_UIMnlAWPushOrPullerGoWidth : UDINT;
	p_UIMnlAWPushOrPullerNomSpd : UDINT;
	p_UIMnlAWPushOrPullerTargetPos : UDINT;
	p_UIMnlAWPushOrPullerStepSize : UDINT;
	p_UIMnlAWPushOrPullerJogSpd : UDINT;
END_VAR
(**)
VAR
	p_UIMnlAWGoWidth : UDINT;
	p_UIMnlAWNomSpd : UDINT;
	p_UIMnlAWTargetPos : UDINT;
	p_UIMnlAWStepSize : UDINT;
	p_UIMnlAWJogSpd : UDINT;
END_VAR
(**)
VAR
	p_UIMnlLifterBtmGoSlt1Pos : UDINT;
	p_UIMnlLifterBtmMag1GoSlt : UDINT;
	p_UIMnlLifterBtmMag2GoSlt : UDINT;
	p_UIMnlLifterBtmMag3GoSlt : UDINT;
	p_UIMnlLifterBtmMag4GoSlt : UDINT;
	p_UIMnlLifterBtmNomSpd : UDINT;
	p_UIMnlLifterBtmTargetPos : UDINT;
	p_UIMnlLifterBtmStepSize : UDINT;
	p_UIMnlLifterBtmJogSpd : UDINT;
END_VAR
(**)
VAR
	p_UIMnlTravNomSpd : UDINT;
	p_UIMnlTravTargetPos : UDINT;
	p_UIMnlTravStepSize : UDINT;
	p_UIMnlTravJogSpd : UDINT;
END_VAR
(**)
VAR
	p_UIVSMEMADSEnA : UDINT;
	p_UIVSMEMADSEnB : UDINT;
	p_UIVSMEMADSBA : UDINT;
	p_UIVSMEMADSBB : UDINT;
END_VAR
(**)
VAR
	p_UILeaderRun : UDINT;
END_VAR
(**)
VAR
	p_UIProdAccData : UDINT;
	p_UIMagAccData : UDINT;
END_VAR
(**)
VAR
	p_UIOpsBypsInitConv : UDINT;
END_VAR
(**)
VAR
	p_UIAIVCommReconnect : UDINT;
END_VAR
(**)
VAR
	p_UINewMag1 : UDINT;
	p_UINewMag2 : UDINT;
	p_UINewMag3 : UDINT;
	p_UINewMag4 : UDINT;
	p_UIRlsMag1 : UDINT;
	p_UIRlsMag2 : UDINT;
	p_UIRlsMag3 : UDINT;
	p_UIRlsMag4 : UDINT;
	p_UIEjectMag1 : UDINT;
	p_UIEjectMag2 : UDINT;
	p_UIEjectMag3 : UDINT;
	p_UIP800Press1 : UDINT;
	p_UIP800Press2 : UDINT;
	p_UIP800Press3 : UDINT;
END_VAR
(**)
VAR
	p_UIAGVSimulateOnline : UDINT;
	p_UIAGVSimulateSig : UDINT;
	p_UIAGVSimulationOn : UDINT;
END_VAR
(**)
VAR
	p_UIMismatchOverWriteConfig : UDINT;
	p_UITempAddrFillDone : UDINT;
	p_UIIPConfigChgDone : UDINT;
	p_UIOverwriteIP : UDINT;
	p_UIOverwriteSubnet : UDINT;
	p_UIOverwriteEthMode : UDINT;
	p_UITeachServo : UDINT;
END_VAR
(**)
VAR
	p_UISOTMagErr1 : UDINT;
	p_UISOTMagErr2 : UDINT;
	p_UISOTMagErr3 : UDINT;
	p_UISOTMagErr4 : UDINT;
	p_UISOTMagRdy1 : UDINT;
	p_UISOTMagRdy2 : UDINT;
	p_UISOTMagRdy3 : UDINT;
	p_UISOTMagRdy4 : UDINT;
	p_UISOTMagAvail1 : UDINT;
	p_UISOTMagAvail2 : UDINT;
	p_UISOTMagAvail3 : UDINT;
	p_UISOTMagAvail4 : UDINT;
	p_UISOTMagSLarge1 : UDINT;
	p_UISOTMagSLarge2 : UDINT;
	p_UISOTMagSLarge3 : UDINT;
	p_UISOTMagSLarge4 : UDINT;
	p_UIAIVReqBring1 : UDINT;
	p_UIAIVReqBring2 : UDINT;
	p_UIAIVReqBring3 : UDINT;
	p_UIAIVReqBring4 : UDINT;
	p_UIAIVReqGet1 : UDINT;
	p_UIAIVReqGet2 : UDINT;
	p_UIAIVReqGet3 : UDINT;
	p_UIAIVReqGet4 : UDINT;
END_VAR
(**)
VAR
	p_UISOTSimulationSig1 : UDINT;
	p_UISOTSimulationSig2 : UDINT;
	p_UISOTSimulationSig3 : UDINT;
	p_UISOTSimulationSig4 : UDINT;
END_VAR
(*USB*)
VAR
	p_UIUSBRun : UDINT;
	p_UIUSBRdrAct : UDINT;
	p_UIResetButton : UDINT;
END_VAR
(**)
VAR
	p_UIMag1SafetyBarAct : UDINT;
	p_UIMag2SafetyBarAct : UDINT;
	p_UIMag3SafetyBarAct : UDINT;
END_VAR
(**)
VAR
	p_UIQueryBoardInfo : UDINT;
	p_UIQueryWorkOrderInfo : UDINT;
	p_UISaveHMIConfigure : UDINT;
	p_UISaveHMISvyConfig : UDINT;
	p_UITopBarcode : UDINT;
	p_UIBottomBarcode : UDINT;
	p_UIMagazineId : UDINT;
	p_UIMagazineSlotId : UDINT;
	p_UIPCBBarcode : UDINT;
	p_UISkipWorkOrder : UDINT;
	p_UIReadWorkOrder : UDINT;
	p_UIDeleteWorkOrder : UDINT;
END_VAR
(**)
VAR
	p_UIUnloadMag : UDINT;
	p_UIBrdOutCntr : UDINT;
END_VAR
(**)
VAR
	p_UIBlkTravLif : UDINT;
END_VAR
(**)
VAR
	p_UIMnlPPNomSpd : UDINT;
	p_UIMnlPPTargetPos : UDINT;
	p_UIMnlPPStepSize : UDINT;
	p_UIMnlPPJogSpd : UDINT;
	p_UISafetyCurtainReset : UDINT;
	p_UIMnlBypCurtainSen : UDINT;
	p_UIMnlBypCurtainPBLED : UDINT;
	p_UIMachineSafetySigToDS : UDINT;
	p_UIHCommModChg : UDINT;
END_VAR
(*Trolley*)
VAR
	p_UITrolleyLckAct1 : UDINT;
	p_UITrolleyLckAct2 : UDINT;
	p_UITrolleyUnlck1 : UDINT;
	p_UITrolleyUnlck2 : UDINT;
END_VAR
(**)
```

### Program Logical/UI/UI (IEC)

#### Init.st - Change By Project
```iecst
(** 2019-03-25 **)
PROGRAM _INIT

	(* Always Change If Project Change *)

	//Pass Address To Global Address For External Use
	//Action, State & Status
	p_UIStat	:= ADR(eStat);
	p_UIStatus	:= ADR(eStatus);
	p_UIStatTxt	:= ADR(sStatTxt);

	//Alarm

	//Output
	p_UIStartupAct 					:= ADR(eStartupAct);
	p_UISimuAct						:= ADR(eSimuAct);
	p_UIHWInfoAct 					:= ADR(eHWInfoAct);
	p_UITLBuzAct 					:= ADR(eTLBuzAct);
	p_UIRstErrAct 					:= ADR(eRstErrAct);
	p_UIProdRcpAct 					:= ADR(eProdRcpAct);
	p_UIMpProdRcpAct				:= ADR(eMpProdRcpAct);
	p_UIMagRcpAct 					:= ADR(eMagRcpAct);
	p_UIMagRcpAct1 					:= ADR(eMagRcpAct1);
	p_UIMcParamAct 					:= ADR(eMcParamAct);
	p_UIUsrMgmtAct 					:= ADR(eUsrMgmtAct);
	p_UIBuffer1Act 					:= ADR(eBuffer1Act);
	p_UIBuffer2Act 					:= ADR(eBuffer2Act);
	p_UIBuffer3Act 					:= ADR(eBuffer3Act);
	p_UIBuffer4Act 					:= ADR(eBuffer4Act);
	p_UIDSSMEMAAAct 				:= ADR(eDSSMEMAAAct);
	p_UIDSSMEMABAct 				:= ADR(eDSSMEMABAct);
	p_UIInShutterAct 				:= ADR(eInShutterAct);
	p_UIInShutterAct2 				:= ADR(eInShutterAct2);
	p_UIInShutterAct3 				:= ADR(eInShutterAct3);
	p_UIOutShutterAct 				:= ADR(eOutShutterAct);
	p_UIOutShutterAct2 				:= ADR(eOutShutterAct2);
	p_UIPullerAct 					:= ADR(ePullerAct);
	p_UIPullConvAct 				:= ADR(ePullConvAct);
	p_UIMagConvSelClp1Act 			:= ADR(eMagConvSelClp1Act);
	p_UIMagConvSelClp2Act 			:= ADR(eMagConvSelClp2Act);
	p_UIMagConvSelClp3Act 			:= ADR(eMagConvSelClp3Act);
	p_UIMagConvSelClp4Act 			:= ADR(eMagConvSelClp4Act);
	p_UIMagConv2Clp1Act 			:= ADR(eMagConv2Clp1Act);
	p_UIMagConv2Clp2Act 			:= ADR(eMagConv2Clp2Act);
	p_UIMagConv2Clp3Act 			:= ADR(eMagConv2Clp3Act);
	p_UIMagConv2Clp4Act 			:= ADR(eMagConv2Clp4Act);
	p_UIServoPPAct 					:= ADR(eServoPullPusherAct);

	p_UIAWPushOrPullerAct 			:= ADR(eAWPushOrPullerAct);
	p_UIAWOpenAct 					:= ADR(eAWOpenAct);
	p_UILifterBtmAct 				:= ADR(eLifterBtmAct);
	p_UITravAct 					:= ADR(eTravAct);
	p_UIDOAct 						:= ADR(eDOAct);
	p_UIHermesAct					:= ADR(eHermesAct);
	p_UILFLeaderAct					:= ADR(eLFLeaderAct);
	p_UIOpsAct						:= ADR(eOpsAct);
	p_UIFrmAct						:= ADR(eFrmAct);
	p_UIMtrPshrAct	 				:= ADR(eMtrPshrAct);

	p_UIMcParamWr					:= ADR(tyMcParamWr);

	p_UIProdRcpInfoIn				:= ADR(tyProdRcpInfoIn);
	p_UIProdRcpSearch				:= ADR(sProdRcpSearch);
	p_UIProdRcpScan					:= ADR(sProdRcpScan);
	p_UIProdRcpCurrRcpWr			:= ADR(tyProdRcpCurrRcpWr);

	p_UIMagRcpInfoIn				:= ADR(tyMagRcpInfoIn);
	p_UIMagRcpSearch				:= ADR(sMagRcpSearch);
	p_UIMagRcpCurrRcpWr				:= ADR(tyMagRcpCurrRcpWr);

	p_UIMagRcpInfoIn1				:= ADR(tyMagRcpInfoIn1);
	p_UIMagRcpSearch1				:= ADR(sMagRcpSearch1);
	p_UIMagRcpCurrRcpWr1			:= ADR(tyMagRcpCurrRcpWr1);

	p_UIUsrMgmtInfoIn				:= ADR(tyUsrMgmtInfoIn);
	p_UIUsrMgmtAccessRightLvl1Wr	:= ADR(tyUsrMgmtAccessRightLvl1Wr);
	p_UIUsrMgmtAccessRightLvl2Wr	:= ADR(tyUsrMgmtAccessRightLvl2Wr);
	p_UIUsrMgmtAccessRightLvl3Wr	:= ADR(tyUsrMgmtAccessRightLvl3Wr);

	p_UIHermesDSParamWr				:= ADR(a_tyHermesDSParamWr);

	P_UISectionLdr					:= ADR(tyP1022McSetVComm.tyLF.tyBtnSectionLdr.bValue);

	p_UISetIPAddr					:= ADR(sSetIPAddr);
	p_UISetSubnetMask				:= ADR(sSetSubnetMask);
	p_UINetworkMode					:= ADR(usiNetworkModeSelected);

	p_UIMnlMod						:= ADR(bManualMod);
	p_UIUIMnlMod					:= ADR(bUIManualMod);
	p_UIMuteBuz						:= ADR(bMuteBuz);
	p_UISimuMod						:= ADR(usiSimuMod);
	p_UINtWr						:= ADR(eNtWr);

	p_UIMnlMtrPshrRetSpd			:= ADR(diMnlMtrPshrExtSpd);
	p_UIMnlMtrPshrRetTorq			:= ADR(diMnlMtrPshrExtTorq);

	p_UIMnlAWPushOrPullerGoWidth	:= ADR(diMnlAWPushOrPullerGoWidth);
	p_UIMnlAWPushOrPullerNomSpd		:= ADR(diMnlAWPushOrPullerNomSpd);
	p_UIMnlAWPushOrPullerTargetPos	:= ADR(diMnlAWPushOrPullerTargetPos);
	p_UIMnlAWPushOrPullerStepSize	:= ADR(diMnlAWPushOrPullerStepSize);
	p_UIMnlAWPushOrPullerJogSpd		:= ADR(diMnlAWPushOrPullerJogSpd);

	p_UIMnlAWGoWidth				:= ADR(diMnlAWGoWidth);
	p_UIMnlAWNomSpd					:= ADR(diMnlAWNomSpd);
	p_UIMnlAWTargetPos				:= ADR(diMnlAWTargetPos);
	p_UIMnlAWStepSize				:= ADR(diMnlAWStepSize);
	p_UIMnlAWJogSpd					:= ADR(diMnlAWJogSpd);

	p_UIMnlLifterBtmGoSlt1Pos		:= ADR(diMnlLifterGoSlt1Pos);
	p_UIMnlLifterBtmMag1GoSlt		:= ADR(diMnlLifterMag1GoSlt);
	p_UIMnlLifterBtmMag2GoSlt		:= ADR(diMnlLifterMag2GoSlt);
	p_UIMnlLifterBtmMag3GoSlt		:= ADR(diMnlLifterMag3GoSlt);
	p_UIMnlLifterBtmMag4GoSlt		:= ADR(diMnlLifterMag4GoSlt);
	p_UIMnlLifterBtmNomSpd			:= ADR(diMnlLifterNomSpd);
	p_UIMnlLifterBtmTargetPos		:= ADR(diMnlLifterTargetPos);
	p_UIMnlLifterBtmStepSize		:= ADR(diMnlLifterStepSize);
	p_UIMnlLifterBtmJogSpd			:= ADR(diMnlLifterJogSpd);

	p_UIMnlTravNomSpd				:= ADR(diMnlTravNomSpd);
	p_UIMnlTravTargetPos			:= ADR(diMnlTravTargetPos);
	p_UIMnlTravStepSize				:= ADR(diMnlTravStepSize);
	p_UIMnlTravJogSpd				:= ADR(diMnlTravJogSpd);

	p_UIVSMEMADSEnA					:= ADR(bVSMEMADSAEn);
	p_UIVSMEMADSEnB					:= ADR(bVSMEMADSBEn);
	p_UIVSMEMADSBA					:= ADR(bVSMEMADSBA);
	p_UIVSMEMADSBB					:= ADR(bVSMEMADSBB);

	p_UILeaderRun					:= ADR(bLeaderRun);

	p_UIProdAccData					:= ADR(bProdAccData);

	p_UIOpsBypsInitConv				:= ADR(bOpsBypsInitConv);

	p_UIAIVCommReconnect			:= ADR(bAIVCommReconnect);

	p_UINewMag1						:= ADR(bNewMag1);
	p_UINewMag2						:= ADR(bNewMag2);
	p_UINewMag3						:= ADR(bNewMag3);
	p_UINewMag4						:= ADR(bNewMag4);
	p_UIRlsMag1						:= ADR(bRlsMag1);
	p_UIRlsMag2						:= ADR(bRlsMag2);
	p_UIRlsMag3						:= ADR(bRlsMag3);
	p_UIRlsMag4						:= ADR(bRlsMag4);
	p_UIEjectMag1					:= ADR(bEjectMag1);
	p_UIEjectMag2					:= ADR(bEjectMag2);
	p_UIEjectMag3					:= ADR(bEjectMag3);
	p_UIP800Press1					:= ADR(tyP0800MagInfo.tyMagInfo1.tyBtnMag1SetEmpty.bValue);
	p_UIP800Press2					:= ADR(tyP0800MagInfo.tyMagInfo1.tyBtnMag2SetEmpty.bValue);
	p_UIP800Press3					:= ADR(tyP0800MagInfo.tyMagInfo2.tyBtnMag3SetEmpty.bValue);

	p_UIAGVSimulateSig		:= ADR(tyAGVSimulateSig);
	p_UIAGVSimulateOnline 	:= ADR(bAGVSimulateOnline);
	p_UIAGVSimulationOn 	:= ADR(bAGVSimulationOn);

	p_UIMismatchOverWriteConfig		:= ADR(bMismatchOverWriteConfig);
	p_UITempAddrFillDone			:= ADR(bTempAddrFillDone);
	p_UIIPConfigChgDone				:= ADR(bIPConfigChgDone);
	p_UIOverwriteIP					:= ADR(bOverwriteIP);
	p_UIOverwriteSubnet				:= ADR(bOverwriteSubnet);
	p_UIOverwriteEthMode			:= ADR(bOverwriteEthMode);

	p_UITeachServo					:= ADR(bTeachServo);

	p_UISOTSimulationSig1 := ADR(tySOTSimulateSig1);
	p_UISOTSimulationSig2 := ADR(tySOTSimulateSig2);
	p_UISOTSimulationSig3 := ADR(tySOTSimulateSig3);
	p_UISOTSimulationSig4 := ADR(tySOTSimulateSig4);

	//AIV Comm
	p_UISOTMagErr1		:= ADR(bSOTMagErr1);
	p_UISOTMagErr2		:= ADR(bSOTMagErr2);
	p_UISOTMagErr3		:= ADR(bSOTMagErr3);
	p_UISOTMagErr4		:= ADR(bSOTMagErr4);
	p_UISOTMagRdy1		:= ADR(bSOTMagRdy1);
	p_UISOTMagRdy2		:= ADR(bSOTMagRdy2);
	p_UISOTMagRdy3		:= ADR(bSOTMagRdy3);
	p_UISOTMagRdy4		:= ADR(bSOTMagRdy4);
	p_UISOTMagAvail1	:= ADR(bSOTMagAvail1);
	p_UISOTMagAvail2	:= ADR(bSOTMagAvail2);
	p_UISOTMagAvail3	:= ADR(bSOTMagAvail3);
	p_UISOTMagAvail4	:= ADR(bSOTMagAvail4);
	p_UISOTMagSLarge1	:= ADR(bSOTMagSLarge1);
	p_UISOTMagSLarge2	:= ADR(bSOTMagSLarge2);
	p_UISOTMagSLarge3	:= ADR(bSOTMagSLarge3);
	p_UISOTMagSLarge4	:= ADR(bSOTMagSLarge4);

	p_UIAIVReqBring1	:= ADR(bAIVReqBring1);
	p_UIAIVReqBring2	:= ADR(bAIVReqBring2);
	p_UIAIVReqBring3	:= ADR(bAIVReqBring3);
	p_UIAIVReqBring4	:= ADR(bAIVReqBring4);
	p_UIAIVReqGet1		:= ADR(bAIVReqGet1);
	p_UIAIVReqGet2		:= ADR(bAIVReqGet2);
	p_UIAIVReqGet3		:= ADR(bAIVReqGet3);
	p_UIAIVReqGet4		:= ADR(bAIVReqGet4);

	p_UIUSBRdrAct		:= ADR(eUSBRdrAct);
	p_UIUSBRun			:= ADR(bUSBRun);
	p_UIResetButton     := ADR(bResetButton);

	p_UIMag1SafetyBarAct:= ADR(eMag1SafetyBarAct);
	p_UIMag2SafetyBarAct:= ADR(eMag2SafetyBarAct);
	p_UIMag3SafetyBarAct:= ADR(eMag3SafetyBarAct);

	p_UIUnloadMag					:= ADR(bUnloadMag);
	p_UIBrdOutCntr 		:= ADR(uiBrdOutCntr); //for LMC opcUA
	p_UIBlkTravLif		:= ADR(bBlkOpsTravLif);

	p_UIMnlAWGoWidth		:= ADR(diMnlAWGoWidth);
	p_UIMnlAWNomSpd			:= ADR(diMnlAWNomSpd);
	p_UIMnlAWTargetPos		:= ADR(diMnlAWTargetPos);
	p_UIMnlAWStepSize		:= ADR(diMnlAWStepSize);
	p_UIMnlAWJogSpd			:= ADR(diMnlAWJogSpd);

	p_UIMnlPPNomSpd				:= ADR(diMnlPPNomSpd);
	p_UIMnlPPTargetPos			:= ADR(diMnlPPTargetPos);
	p_UIMnlPPStepSize			:= ADR(diMnlPPStepSize);
	p_UIMnlPPJogSpd				:= ADR(diMnlPPJogSpd);

	p_UISafetyCurtainReset		:= ADR(bSafetyCurtainReset);
	p_UIMnlBypCurtainPBLED		:= ADR(bBypCurtainPBLED);
	p_UIMnlBypCurtainSen		:= ADR(bBypCurtainSen);
	p_UIMachineSafetySigToDS 	:= ADR(bMachineSafetySigToDS);

	//new for Hermes 1.3
	p_UIHermesSvyParamWr			:= ADR(tyHermesSvyParamWr);
	p_UIQueryBoardInfo				:= ADR(bQueryBoardInfo);
	p_UIQueryWorkOrderInfo			:= ADR(bQueryWorkOrderInfo);
	p_UISaveHMIConfigure            := ADR(bSaveHMIConfigure);
	p_UISaveHMISvyConfig            := ADR(bSaveHMISvyConfig);
	p_UITopBarcode                  := ADR(tyP0201OpsTravLifter.tyQueryBoardInfo.tyStringTopBarcode.sValue);
	p_UIBottomBarcode               := ADR(tyP0201OpsTravLifter.tyQueryBoardInfo.tyStringBottomBarcode.sValue);
	p_UIMagazineId                  := ADR(tyP0201OpsTravLifter.tyQueryWorkOrderInfo.tyStringMagazineId.sValue);
	p_UIMagazineSlotId              := ADR(iSlotId);
	p_UIPCBBarcode                  := ADR(tyP0201OpsTravLifter.tyQueryWorkOrderInfo.tyStringBarcode.sValue);
	p_UISkipWorkOrder		    	:= ADR(bSkipWorkOrder);
	p_UIReadWorkOrder		    	:= ADR(bReadWorkOrder);
	p_UIDeleteWorkOrder		    	:= ADR(bDeleteWorkOrder);
	//Horizontal comm
	p_UIHCommModChg					:= ADR(bHCommModChg);

	p_UITrolleyLckAct1				:= ADR(eTrolleyLckAct1);
	p_UITrolleyLckAct2				:= ADR(eTrolleyLckAct2);
	p_UITrolleyUnlck1				:= ADR(tyP0200OpsGen.tyOps.tyBtnTrolleyUnlck1.bValue);
	p_UITrolleyUnlck2				:= ADR(tyP0200OpsGen.tyOps.tyBtnTrolleyUnlck2.bValue);

END_PROGRAM
```

#### Act_InitGlobal.st - Change By Project
```iecst
(** 2019-03-25 **)
ACTION Act_InitGlobal:

	//Pass Data To Internal Use
	p_eAct ACCESS p_StartupUIAct;

	p_bOpsRun ACCESS p_OpsRun;

	p_bStartupRun ACCESS p_StartupRun;
	p_eStartupStat ACCESS p_StartupStat;
	p_eStartupStatus ACCESS p_StartupStatus;
	p_sStartupStatTxt ACCESS p_StartupStatTxt;
	p_eStartupStep ACCESS p_StartupStep;
	p_sStartupStepTxt ACCESS p_StartupStepTxt;
	p_bStartupGetConfigDone ACCESS p_StartupGetConfigDone;
	p_bStartupMismatchSetConfigDone ACCESS p_StartupMismatchSetConfigDone;
	p_bStartupUISettingsLoadDone ACCESS p_StartupUISettingsLoadDone;

	p_eHWInfoStat ACCESS p_HWInfoStat;
	p_eHWInfoStatus ACCESS p_HWInfoStatus;
	p_sHWInfoStatTxt ACCESS p_HWInfoStatTxt;
	p_sHWInfoIPAddr ACCESS p_HWInfoIPAddr;
	p_sHWInfoSubnetMask ACCESS p_HWInfoSubnetMask;
	p_udiHWInfoEthMode ACCESS p_HWInfoEthMode;

	p_eTLBuzStat ACCESS p_TLBuzStat;
	p_eTLBuzStatus ACCESS p_TLBuzStatus;
	p_sTLBuzStatTxt ACCESS p_TLBuzStatTxt;

	p_tyAlarmCurrList ACCESS p_AlarmCurrList;
	p_tyAlarmRcyList ACCESS p_AlarmRecoveryList;
	p_tyAlarmHistoryList ACCESS p_AlarmHistoryList;
	p_bAlarmWarning ACCESS p_AlarmWarning;
	p_bAlarmErr ACCESS p_AlarmErr;
	p_bAlarmInfo ACCESS p_AlarmInfo;
	p_bAlarmInfoLF ACCESS p_AlarmInfoLF;
	p_sAlarmInfoMsg ACCESS p_AlarmInfoMsg;

	p_eRstErrStat ACCESS p_RstErrStat;
	p_eRstErrStatus ACCESS p_RstErrStatus;
	p_sRstErrStatTxt ACCESS p_RstErrStatTxt;

	p_eProdRcpStat ACCESS p_ProdRcpStat;
	p_eProdRcpStatus ACCESS p_ProdRcpStatus;
	p_sProdRcpStatTxt ACCESS p_ProdRcpStatTxt;
	p_tyProdRcpFilterList ACCESS p_ProdRcpFilterList;
	p_tyProdRcpSortedList ACCESS p_ProdRcpSortedList;
	p_tyProdRcpCurrList	ACCESS p_ProdRcpCurrList;
	p_tyProdRcpCurrRcp0 ACCESS p_ProdRcpCurrRcp0;
	p_tyProdRcpCurrRcp1 ACCESS p_ProdRcpCurrRcp1;
	p_tyProdRcpCurrRcp2 ACCESS p_ProdRcpCurrRcp2;
	p_tyProdRcpInfoOut ACCESS p_ProdRcpInfoOut;
	p_bProdRcpNmEmpty ACCESS p_ProdRcpNmEmpty;
	p_bProdRcpListFull ACCESS p_ProdRcpListFull;
	p_bProdRcpNmNotExist ACCESS p_ProdRcpNmNotExist;

	p_eMpProdRcpStat ACCESS p_MpProdRcpStat;
	p_eMpProdRcpStatus ACCESS p_MpProdRcpStatus;

	p_eMagRcpStat ACCESS p_MagRcpStat;
	p_eMagRcpStatus ACCESS p_MagRcpStatus;
	p_sMagRcpStatTxt ACCESS p_MagRcpStatTxt;
	p_tyMagRcpFilterList ACCESS p_MagRcpFilterList;
	p_tyMagRcpSortedList ACCESS p_MagRcpSortedList;
	p_tyMagRcpCurrList ACCESS p_MagRcpCurrList;
	p_tyMagRcpInfoOut ACCESS p_MagRcpInfoOut;
	p_tyMagRcpCurrRcp ACCESS p_MagRcpCurrRcp;
	p_bMagRcpNmEmpty ACCESS p_MagRcpNmEmpty;
	p_bMagRcpListFull ACCESS p_MagRcpListFull;
	p_bMagRcpNmNotExist ACCESS p_MagRcpNmNotExist;

	p_eMagRcpStat1 ACCESS p_MagRcpStat1;
	p_eMagRcpStatus1 ACCESS p_MagRcpStatus1;
	p_sMagRcpStatTxt1 ACCESS p_MagRcpStatTxt1;
	p_tyMagRcpFilterList1 ACCESS p_MagRcpFilterList1;
	p_tyMagRcpSortedList1 ACCESS p_MagRcpSortedList1;
	p_tyMagRcpCurrList1 ACCESS p_MagRcpCurrList1;
	p_tyMagRcpInfoOut1 ACCESS p_MagRcpInfoOut1;
	p_tyMagRcpCurrRcp1 ACCESS p_MagRcpCurrRcp1;
	p_bMagRcpNmEmpty1 ACCESS p_MagRcpNmEmpty1;
	p_bMagRcpListFull1 ACCESS p_MagRcpListFull1;
	p_bMagRcpNmNotExist1 ACCESS p_MagRcpNmNotExist1;
	p_diMagRcp1TravPos ACCESS p_MagRcpCurrRcpMag1TravPos;
	p_diMagRcp2TravPos ACCESS p_MagRcpCurrRcpMag2TravPos;
	p_diMagRcp3TravPos ACCESS p_MagRcpCurrRcpMag3TravPos;

	p_eMcParamStat ACCESS p_McParamStat;
	p_eMcParamStatus ACCESS p_McParamStatus;
	p_sMcParamStatTxt ACCESS p_McParamStatTxt;
	p_tyMcParamCurr	ACCESS p_McParamCurr;

	p_tyNtParamCurr ACCESS p_NtParamCurr;

	p_eUsrMgmtStat ACCESS p_UsrMgmtStat;
	p_eUsrMgmtStatus ACCESS p_UsrMgmtStatus;
	p_sUsrMgmtStatTxt ACCESS p_UsrMgmtStatTxt;
	p_tyUsrMgmtCurrUsr ACCESS p_UsrMgmtCurrUsr;
	p_tyUsrMgmtCurrAccessRgt ACCESS p_UsrMgmtCurrAccessRight;
	p_tyUsrMgmtAllList ACCESS p_UsrMgmtAllList;
	p_tyUsrMgmtLv2List ACCESS p_UsrMgmtLvl2List;
	p_tyUsrMgmtLv3List ACCESS p_UsrMgmtLvl3List;
	p_tyUsrMgmtAdminList ACCESS p_UsrMgmtAdminList;
	p_bUsrMgmtNmEmpty ACCESS p_UsrMgmtNmEmpty;
	p_bUsrMgmtListFull ACCESS p_UsrMgmtListFull;
	p_bUsrMgmtNmExist ACCESS p_UsrMgmtNmExist;
	p_bUsrMgmtNmNotExist ACCESS p_UsrMgmtNmNotExist;
	p_bUsrMgmtLastAdmin ACCESS p_UsrMgmtLastAdmin;
	p_bUsrMgmtLoginSuccess ACCESS p_UsrMgmtLoginSuccess;
	p_bUsrMgmtPwMismatch ACCESS p_UsrMgmtPwMismatch;
	p_bUsrMgmtUnableDelete ACCESS p_UsrMgmtUnableDelete;
	p_tyUsrMgmtFullData ACCESS p_UsrMgmtFullData;

	p_eBuffer1Stat ACCESS p_Buffer1Stat;
	p_eBuffer1Status ACCESS p_Buffer1Status;
	p_sBuffer1StatTxt ACCESS p_Buffer1StatTxt;
	p_tyBuffer1DispBffr ACCESS p_Buffer1DispBffr;
	p_tyBuffer1BffrStat ACCESS p_Buffer1BffrStat;
	p_bBuffer1MagPresent ACCESS p_Buffer1MagPresent;
	p_bBuffer1MagRemoved ACCESS p_Buffer1MagRemoved;

	p_eBuffer2Stat ACCESS p_Buffer2Stat;
	p_eBuffer2Status ACCESS p_Buffer2Status;
	p_sBuffer2StatTxt ACCESS p_Buffer2StatTxt;
	p_tyBuffer2DispBffr ACCESS p_Buffer2DispBffr;
	p_tyBuffer2BffrStat ACCESS p_Buffer2BffrStat;
	p_bBuffer2MagPresent ACCESS p_Buffer2MagPresent;
	p_bBuffer2MagRemoved ACCESS p_Buffer2MagRemoved;

	p_eBuffer3Stat ACCESS p_Buffer3Stat;
	p_eBuffer3Status ACCESS p_Buffer3Status;
	p_sBuffer3StatTxt ACCESS p_Buffer3StatTxt;
	p_tyBuffer3DispBffr ACCESS p_Buffer3DispBffr;
	p_tyBuffer3BffrStat ACCESS p_Buffer3BffrStat;
	p_bBuffer3MagPresent ACCESS p_Buffer3MagPresent;
	p_bBuffer3MagRemoved ACCESS p_Buffer3MagRemoved;

	p_eBuffer4Stat ACCESS p_Buffer4Stat;
	p_eBuffer4Status ACCESS p_Buffer4Status;
	p_sBuffer4StatTxt ACCESS p_Buffer4StatTxt;
	p_tyBuffer4DispBffr ACCESS p_Buffer4DispBffr;
	p_tyBuffer4BffrStat ACCESS p_Buffer4BffrStat;
	p_bBuffer4MagPresent ACCESS p_Buffer4MagPresent;
	p_bBuffer4MagRemoved ACCESS p_Buffer4MagRemoved;

	p_eDSSMEMAAStat ACCESS p_DSSMEMAAStat;
	p_eDSSMEMAAStatus ACCESS p_DSSMEMAAStatus;
	p_sDSSMEMAAStatTxt ACCESS p_DSSMEMAAStatTxt;
	p_bDSSMEMAAUSRdy ACCESS p_DSSMEMAAUSRdy;
	p_bDSSMEMAAUSGdBrdRdy ACCESS p_DSSMEMAAUSGdBrdRdy;
	p_bDSSMEMAADSRdy ACCESS p_DSSMEMAADSRdy;

	p_eDSSMEMABStat ACCESS p_DSSMEMABStat;
	p_eDSSMEMABStatus ACCESS p_DSSMEMABStatus;
	p_sDSSMEMABStatTxt ACCESS p_DSSMEMABStatTxt;
	p_bDSSMEMABUSRdy ACCESS p_DSSMEMABUSRdy;
	p_bDSSMEMABUSGdBrdRdy ACCESS p_DSSMEMABUSGdBrdRdy;
	p_bDSSMEMABDSRdy ACCESS p_DSSMEMABDSRdy;

	p_eInShutterStat ACCESS p_Pneu2SenInShutterStat;
	p_eInShutterStatus ACCESS p_Pneu2SenInShutterStatus;
	p_sInShutterStatTxt ACCESS p_Pneu2SenInShutterStatTxt;
	p_bInShutterExtCtrl ACCESS p_Pneu2SenInShutterExtCtrl;
	p_bInShutterRetCtrl ACCESS p_Pneu2SenInShutterRetCtrl;
	p_bInShutterTwoCtrlOut ACCESS p_Pneu2SenInShutterTwoCtrlOut;
	p_bInShutterExtended ACCESS p_Pneu2SenInShutterExtended;
	p_bInShutterRetracted ACCESS p_Pneu2SenInShutterRetracted;

	p_eInShutterStat2 ACCESS p_Pneu2SenInShutterStat2;
	p_eInShutterStatus2 ACCESS p_Pneu2SenInShutterStatus2;
	p_sInShutterStatTxt2 ACCESS p_Pneu2SenInShutterStatTxt2;
	p_bInShutterExtCtrl2 ACCESS p_Pneu2SenInShutterExtCtrl2;
	p_bInShutterRetCtrl2 ACCESS p_Pneu2SenInShutterRetCtrl2;
	p_bInShutterTwoCtrlOut2 ACCESS p_Pneu2SenInShutterTwoCtrlOut2;
	p_bInShutterExtended2 ACCESS p_Pneu2SenInShutterExtended2;
	p_bInShutterRetracted2 ACCESS p_Pneu2SenInShutterRetracted2;

	p_eInShutterStat3 ACCESS p_Pneu2SenInShutterStat3;
	p_eInShutterStatus3 ACCESS p_Pneu2SenInShutterStatus3;
	p_sInShutterStatTxt3 ACCESS p_Pneu2SenInShutterStatTxt3;
	p_bInShutterExtCtrl3 ACCESS p_Pneu2SenInShutterExtCtrl3;
	p_bInShutterRetCtrl3 ACCESS p_Pneu2SenInShutterRetCtrl3;
	p_bInShutterTwoCtrlOut3 ACCESS p_Pneu2SenInShutterTwoCtrlOut3;
	p_bInShutterExtended3 ACCESS p_Pneu2SenInShutterExtended3;
	p_bInShutterRetracted3 ACCESS p_Pneu2SenInShutterRetracted3;

	p_eOutShutterStat ACCESS p_Pneu2SenOutShutterStat;
	p_eOutShutterStatus ACCESS p_Pneu2SenOutShutterStatus;
	p_sOutShutterStatTxt ACCESS p_Pneu2SenOutShutterStatTxt;
	p_bOutShutterExtCtrl ACCESS p_Pneu2SenOutShutterExtCtrl;
	p_bOutShutterRetCtrl ACCESS p_Pneu2SenOutShutterRetCtrl;
	p_bOutShutterTwoCtrlOut ACCESS p_Pneu2SenOutShutterTwoCtrlOut;
	p_bOutShutterExtended ACCESS p_Pneu2SenOutShutterExtended;
	p_bOutShutterRetracted ACCESS p_Pneu2SenOutShutterRetracted;

	p_eOutShutterStat2 ACCESS p_Pneu2SenOutShutterStat2;
	p_eOutShutterStatus2 ACCESS p_Pneu2SenOutShutterStatus2;
	p_sOutShutterStatTxt2 ACCESS p_Pneu2SenOutShutterStatTxt2;
	p_bOutShutterExtCtrl2 ACCESS p_Pneu2SenOutShutterExtCtrl2;
	p_bOutShutterRetCtrl2 ACCESS p_Pneu2SenOutShutterRetCtrl2;
	p_bOutShutterTwoCtrlOut2 ACCESS p_Pneu2SenOutShutterTwoCtrlOut2;
	p_bOutShutterExtended2 ACCESS p_Pneu2SenOutShutterExtended2;
	p_bOutShutterRetracted2 ACCESS p_Pneu2SenOutShutterRetracted2;

	p_eSelClamp1Stat ACCESS p_PneuNoSenSelClamp1Stat;
	p_eSelClamp1Status ACCESS p_PneuNoSenSelClamp1Status;
	p_sSelClamp1StatTxt ACCESS p_PneuNoSenSelClamp1StatTxt;
	p_bSelClamp1ExtCtrl ACCESS p_PneuNoSenSelClamp1ExtCtrl;
	p_bSelClamp1RetCtrl ACCESS p_PneuNoSenSelClamp1RetCtrl;
	p_bSelClamp1TwoCtrlOut ACCESS p_PneuNoSenSelClamp1TwoCtrlOut;
	p_bSelClamp1Extended ACCESS p_PneuNoSenSelClamp1Extended;
	p_bSelClamp1Retracted ACCESS p_PneuNoSenSelClamp1Retracted;

	p_eSelClamp2Stat ACCESS p_PneuNoSenSelClamp2Stat;
	p_eSelClamp2Status ACCESS p_PneuNoSenSelClamp2Status;
	p_sSelClamp2StatTxt ACCESS p_PneuNoSenSelClamp2StatTxt;
	p_bSelClamp2ExtCtrl ACCESS p_PneuNoSenSelClamp2ExtCtrl;
	p_bSelClamp2RetCtrl ACCESS p_PneuNoSenSelClamp2RetCtrl;
	p_bSelClamp2TwoCtrlOut ACCESS p_PneuNoSenSelClamp2TwoCtrlOut;
	p_bSelClamp2Extended ACCESS p_PneuNoSenSelClamp2Extended;
	p_bSelClamp2Retracted ACCESS p_PneuNoSenSelClamp2Retracted;

	p_eSelClamp3Stat ACCESS p_PneuNoSenSelClamp3Stat;
	p_eSelClamp3Status ACCESS p_PneuNoSenSelClamp3Status;
	p_sSelClamp3StatTxt ACCESS p_PneuNoSenSelClamp3StatTxt;
	p_bSelClamp3ExtCtrl ACCESS p_PneuNoSenSelClamp3ExtCtrl;
	p_bSelClamp3RetCtrl ACCESS p_PneuNoSenSelClamp3RetCtrl;
	p_bSelClamp3TwoCtrlOut ACCESS p_PneuNoSenSelClamp3TwoCtrlOut;
	p_bSelClamp3Extended ACCESS p_PneuNoSenSelClamp3Extended;
	p_bSelClamp3Retracted ACCESS p_PneuNoSenSelClamp3Retracted;

	p_eSelClamp4Stat ACCESS p_PneuNoSenSelClamp4Stat;
	p_eSelClamp4Status ACCESS p_PneuNoSenSelClamp4Status;
	p_sSelClamp4StatTxt ACCESS p_PneuNoSenSelClamp4StatTxt;
	p_bSelClamp4ExtCtrl ACCESS p_PneuNoSenSelClamp4ExtCtrl;
	p_bSelClamp4RetCtrl ACCESS p_PneuNoSenSelClamp4RetCtrl;
	p_bSelClamp4TwoCtrlOut ACCESS p_PneuNoSenSelClamp4TwoCtrlOut;
	p_bSelClamp4Extended ACCESS p_PneuNoSenSelClamp4Extended;
	p_bSelClamp4Retracted ACCESS p_PneuNoSenSelClamp4Retracted;

	p_ePullerStat ACCESS p_Pneu2SenPullerStat;
	p_ePullerStatus ACCESS p_Pneu2SenPullerStatus;
	p_sPullerStatTxt ACCESS p_Pneu2SenPullerStatTxt;
	p_bPullerExtCtrl ACCESS p_Pneu2SenPullerExtCtrl;
	p_bPullerRetCtrl ACCESS p_Pneu2SenPullerRetCtrl;
	p_bPullerTwoCtrlOut ACCESS p_Pneu2SenPullerTwoCtrlOut;
	p_bPullerExtended ACCESS p_Pneu2SenPullerExtended;
	p_bPullerRetracted ACCESS p_Pneu2SenPullerRetracted;

	p_ePullConvStat ACCESS p_PullConvStat;
	p_ePullConvStatus ACCESS p_PullConvStatus;
	p_sPullConvStatTxt ACCESS p_PullConvStatTxt;
	p_bPullConvHvBrd ACCESS p_PullConvHvBrd;
	p_bPullConvGdBrd ACCESS p_PullConvGdBrd;
	p_bPullConvMtrSigOnOrLToR ACCESS p_PullConvMtrSigOnOrLToR;
	p_bPullConvMtrDirOrRToL ACCESS p_PullConvMtrDirOrRToL;
	p_bPullConvPullerExtCtrl ACCESS p_PullConvPullerExtCtrl;
	p_bPullConvPullerRetCtrl ACCESS p_PullConvPullerRetCtrl;
	p_bPullConvPullerTwoOutputCtrl ACCESS p_PullConvPullerTwoOutputControl;
	p_bPullConvRotRemoteCtrl ACCESS p_PullConvRotRemoteCtrl;
	p_bPullConvRotTwoOutputCtrl ACCESS p_PullConvRotTwoOutputControl;

	p_eMagConv2Clp1Stat ACCESS p_MagConv2Clp1Stat;
	p_eMagConv2Clp1Status ACCESS p_MagConv2Clp1Status;
	p_sMagConv2Clp1StatTxt ACCESS p_MagConv2Clp1StatTxt;
	p_bMagConv2Clp1HvMag ACCESS p_MagConv2Clp1HvMag;
	p_bMagConv2Clp1MtrSigOnOrLToR ACCESS p_MagConv2Clp1MtrSigOnOrLToR;
	p_bMagConv2Clp1MtrDirOrRToL ACCESS p_MagConv2Clp1MtrDirOrRToL;
	p_bMagConv2Clp1ClprFixClampCtrl ACCESS p_MagConv2Clp1FixClprClampCtrl;
	p_bMagConv2Clp1ClprRmtClampCtrl ACCESS p_MagConv2Clp1RmtClprClampCtrl;
	p_bMagConv2Clp1ClprTwoOutputCtrl ACCESS p_MagConv2Clp1ClprTwoOutputCtrl;

	p_eMagConv2Clp2Stat ACCESS p_MagConv2Clp2Stat;
	p_eMagConv2Clp2Status ACCESS p_MagConv2Clp2Status;
	p_sMagConv2Clp2StatTxt ACCESS p_MagConv2Clp2StatTxt;
	p_bMagConv2Clp2HvMag ACCESS p_MagConv2Clp2HvMag;
	p_bMagConv2Clp2MtrSigOnOrLToR ACCESS p_MagConv2Clp2MtrSigOnOrLToR;
	p_bMagConv2Clp2MtrDirOrRToL ACCESS p_MagConv2Clp2MtrDirOrRToL;
	p_bMagConv2Clp2ClprFixClampCtrl ACCESS p_MagConv2Clp2FixClprClampCtrl;
	p_bMagConv2Clp2ClprRmtClampCtrl ACCESS p_MagConv2Clp2RmtClprClampCtrl;
	p_bMagConv2Clp2ClprTwoOutputCtrl ACCESS p_MagConv2Clp2ClprTwoOutputCtrl;

	p_eMagConv2Clp3Stat ACCESS p_MagConv2Clp3Stat;
	p_eMagConv2Clp3Status ACCESS p_MagConv2Clp3Status;
	p_sMagConv2Clp3StatTxt ACCESS p_MagConv2Clp3StatTxt;
	p_bMagConv2Clp3HvMag ACCESS p_MagConv2Clp3HvMag;
	p_bMagConv2Clp3MtrSigOnOrLToR ACCESS p_MagConv2Clp3MtrSigOnOrLToR;
	p_bMagConv2Clp3MtrDirOrRToL ACCESS p_MagConv2Clp3MtrDirOrRToL;
	p_bMagConv2Clp3ClprFixClampCtrl ACCESS p_MagConv2Clp3FixClprClampCtrl;
	p_bMagConv2Clp3ClprRmtClampCtrl ACCESS p_MagConv2Clp3RmtClprClampCtrl;
	p_bMagConv2Clp3ClprTwoOutputCtrl ACCESS p_MagConv2Clp3ClprTwoOutputCtrl;

	p_eMagConv2Clp4Stat ACCESS p_MagConv2Clp4Stat;
	p_eMagConv2Clp4Status ACCESS p_MagConv2Clp4Status;
	p_sMagConv2Clp4StatTxt ACCESS p_MagConv2Clp4StatTxt;
	p_bMagConv2Clp4HvMag ACCESS p_MagConv2Clp4HvMag;
	p_bMagConv2Clp4MtrSigOnOrLToR ACCESS p_MagConv2Clp4MtrSigOnOrLToR;
	p_bMagConv2Clp4MtrDirOrRToL ACCESS p_MagConv2Clp4MtrDirOrRToL;
	p_bMagConv2Clp4ClprFixClampCtrl ACCESS p_MagConv2Clp4FixClprClampCtrl;
	p_bMagConv2Clp4ClprRmtClampCtrl ACCESS p_MagConv2Clp4RmtClprClampCtrl;
	p_bMagConv2Clp4ClprTwoOutputCtrl ACCESS p_MagConv2Clp4ClprTwoOutputCtrl;

	p_bAWPushOrPullerPrep ACCESS p_NtParamAWPusherPrep;
	p_eAWPushOrPullerStat ACCESS p_AWPushOrPullerStat;
	p_eAWPushOrPullerStatus ACCESS p_AWPushOrPullerStatus;
	p_sAWPushOrPullerStatTxt ACCESS p_AWPushOrPullerStatTxt;
	p_udiAWPushOrPullerAxisErrID ACCESS p_AWPushOrPullerAxisErrID;
	p_bAWPushOrPullerAxisErr ACCESS p_AWPushOrPullerAxisErr;
	p_bAWPushOrPullerPwrOn ACCESS p_AWPushOrPullerPwrOn;
	p_bAWPushOrPullerIsHomed ACCESS p_AWPushOrPullerIsHomed;
	p_diAWPushOrPullerActualPos ACCESS p_AWPushOrPullerActualPos;
	p_bAWPushOrPullerFwdLmtSen ACCESS p_AWPushOrPullerFwdLmtSen;
	p_bAWPushOrPullerRevLmtSen ACCESS p_AWPushOrPullerRevLmtSen;
	p_sAWPushOrPullerAxisErrTxt ACCESS p_AWPushOrPullerAxisErrTxt;
	p_bAWPushOrPullerJogging ACCESS p_AWPushOrPullerJogging;
	p_bAWPushOrPullerOpenSen ACCESS p_AWPushOrPullerOpenSen;
	p_bAWPushOrPullerCloseSen ACCESS p_AWPushOrPullerCloseSen;

	p_eAWOpenStat ACCESS p_AWOpenStat;
	p_eAWOpenStatus ACCESS p_AWOpenStatus;
	p_sAWOpenStatTxt ACCESS p_AWOpenStatTxt;
	p_udiAWOpenAxisErrID ACCESS p_AWOpenAxisErrID;
	p_bAWOpenAxisErr ACCESS p_AWOpenAxisErr;
	p_bAWOpenPwrOn ACCESS p_AWOpenPwrOn;
	p_bAWOpenIsHomed ACCESS p_AWOpenIsHomed;
	p_diAWOpenActualPos ACCESS p_AWOpenActualPos;
	p_bAWOpenFwdLmtSen ACCESS p_AWOpenFwdLmtSen;
	p_bAWOpenRevLmtSen ACCESS p_AWOpenRevLmtSen;
	p_bAWOpenWidthPosDiff ACCESS p_AWOpenWidthPosDiff;
	p_sAWOpenAxisErrTxt ACCESS p_AWOpenAxisErrTxt;
	p_bAWOpenJogging ACCESS p_AWOpenJogging;
	p_bAWOpenOpenSen ACCESS p_AWOpenOpenSen;
	p_bAWOpenCloseSen ACCESS p_AWOpenCloseSen;

	p_eLifterBtmStat ACCESS p_LifterBtmStat;
	p_eLifterBtmStatus ACCESS p_LifterBtmStatus;
	p_sLifterBtmStatTxt ACCESS p_LifterBtmStatTxt;
	p_bLifterBtmPwrOn ACCESS p_LifterBtmPwrOn;
	p_bLifterBtmIsHomed ACCESS p_LifterBtmIsHomed;
	p_bLifterBtmPosDiff ACCESS p_LifterBtmPosDiff;
	p_bLifterBtmAxisErr ACCESS p_LifterBtmAxisErr;
	p_udiLifterBtmAxisErrID ACCESS p_LifterBtmAxisErrID;
	p_sLifterBtmAxisErrTxt ACCESS p_LifterBtmAxisErrTxt;
	p_bLifterBtmFwdLmtSen ACCESS p_LifterBtmFwdLmtSen;
	p_bLifterBtmRevLmtSen ACCESS p_LifterBtmRevLmtSen;
	p_diLifterBtmActualPos ACCESS p_LifterBtmActualPos;
	p_bLifterBtmJogging ACCESS p_LifterBtmJogging;
	p_diLifterBtmCurrSltA ACCESS p_LifterBtmCurrSltA;
	p_diLifterBtmCurrSltB ACCESS p_LifterBtmCurrSltB;
	p_diLifterBtmCurrSltC ACCESS p_LifterBtmCurrSltC;
	p_bLifterBtmUpSen ACCESS p_LifterBtmUpSen;
	p_bLifterBtmDownSen ACCESS p_LifterBtmDownSen;
	p_bLifterBtmSltAPosDiff ACCESS p_LifterBtmSltAPosDiff;

	p_eTravStat ACCESS p_TravStat;
	p_eTravStatus ACCESS p_TravStatus;
	p_sTravStatTxt	ACCESS p_TravStatTxt;
	p_bTravPwrOn ACCESS p_TravPwrOn;
	p_bTravIsHomed ACCESS p_TravIsHomed;
	p_bTravPosDiff ACCESS p_TravPosDiff;
	p_bTravAxisErr ACCESS p_TravAxisErr;
	p_udiTravAxisErrID ACCESS p_TravAxisErrID;
	p_sTravAxisErrTxt ACCESS p_TravAxisErrTxt;
	p_bTravFwdLmtSen ACCESS p_TravFwdLmtSen;
	p_bTravRevLmtSen ACCESS p_TravRevLmtSen;
	p_diTravActualPos ACCESS p_TravActualPos;
	p_bTravJogging ACCESS p_TravJogging;
	p_bTravFrontSen ACCESS p_TravFrontSen;
	p_bTravRearSen ACCESS p_TravRearSen;
	p_bTravAPosDiff ACCESS p_TravAPosDiff;
	p_bTravBPosDiff ACCESS p_TravBPosDiff;
	p_bTravCPosDiff ACCESS p_TravCPosDiff;
	p_bTravDPosDiff ACCESS p_TravDPosDiff;
	p_bTravEPosDiff ACCESS p_TravEPosDiff;
	p_bTravFPosDiff ACCESS p_TravFPosDiff;
	p_bTravGPosDiff ACCESS p_TravGPosDiff;
	p_bTravHPosDiff ACCESS p_TravHPosDiff;

	p_tyDI ACCESS p_DI;

	p_eDOStat ACCESS p_DOStat;
	p_eDOStatus ACCESS p_DOStatus;
	p_sDOStatTxt ACCESS p_DOStatTxt;
	p_tyDO ACCESS p_DO;

	p_eHermesStat ACCESS p_HermesStat;
	p_eHermesStatus ACCESS p_HermesStatus;
	p_tyHermesConfiguration ACCESS p_HermesConfiguration;

	p_eDSHermesAStat ACCESS p_DSHermesAStat;
	p_eDSHermesAStatus ACCESS p_DSHermesAStatus;
	p_sDSHermesAStatTxt ACCESS p_DSHermesAStatTxt;
	p_bDSHermesAUSRdy ACCESS p_DSHermesAUSRdy;
	p_bDSHermesADSRdy ACCESS p_DSHermesADSRdy;
	p_bDSHermesAUSGdRdy ACCESS p_DSHermesAUSGdRdy;
	p_bDSHermesADSGdRdy ACCESS p_DSHermesADSGdRdy;
	p_bDSHermesAConnected ACCESS p_DSHermesAConnected;

	p_eDSHermesBStat ACCESS p_DSHermesBStat;
	p_eDSHermesBStatus ACCESS p_DSHermesBStatus;
	p_sDSHermesBStatTxt ACCESS p_DSHermesBStatTxt;
	p_bDSHermesBUSRdy ACCESS p_DSHermesBUSRdy;
	p_bDSHermesBDSRdy ACCESS p_DSHermesBDSRdy;
	p_bDSHermesBUSGdRdy ACCESS p_DSHermesBUSGdRdy;
	p_bDSHermesBDSGdRdy ACCESS p_DSHermesBDSGdRdy;
	p_bDSHermesBConnected ACCESS p_DSHermesBConnected;

	p_eLFLeaderStat ACCESS p_LFLeaderStat;
	p_eLFLeaderStatus ACCESS p_LFLeaderStatus;
	p_tyLFLeaderFollowerInfo ACCESS p_LFLeaderFollowerInfo;
	p_tyLFLeaderFollowerToLeaderTag ACCESS p_LFLeaderFollowerToLeaderTag;

	p_bLFFollowerProdAccDataMnl ACCESS p_LFFollowerProdAccDataMnl;
	p_bLFFollowerLdrSeqCtrlInActive ACCESS p_LFFollowerLdrSeqCtrlInActive;
	p_bLFFollowerDSAllow ACCESS p_LFFollowerDSAllow;
	p_bLFFollowerUSAllow ACCESS p_LFFollowerUSAllow;

	p_bLCSLFAccDataMnl ACCESS p_LCSLFAccDataMnl;

	p_eOpsStat ACCESS p_OpsStat;
	p_eOpsStatus ACCESS p_OpsStatus;
	p_sOpsStatTxt ACCESS p_OpsStatTxt;
	p_eOpsOpsStatus ACCESS p_OpsOpsStatus;
	p_bOpsStatusRun ACCESS p_OpsStatusRun;
	p_bOpsStatusStop ACCESS p_OpsStatusStop;
	p_bOpsStatusCycleStop ACCESS p_OpsStatusCycleStop;
	p_bOpsStatusStep ACCESS p_OpsStatusStep;

	p_sOpsTravLifLDStepTxt ACCESS p_OpsTravLifLDStepTxt;
	//	p_sOpsMagLD1StepTxt ACCESS p_OpsMagLD1StepTxt;
	//	p_sOpsMagLD2StepTxt ACCESS p_OpsMagLD2StepTxt;
	//	p_sOpsMagLD3StepTxt ACCESS p_OpsMagLD3StepTxt;
	//	p_sOpsMagLD4StepTxt ACCESS p_OpsMagLD4StepTxt;
	p_sOpsMagConvLD1StepTxt ACCESS p_OpsMagConvLD1StepTxt;
	p_sOpsMagConvLD2StepTxt ACCESS p_OpsMagConvLD2StepTxt;
	p_sOpsMagConvLD3StepTxt ACCESS p_OpsMagConvLD3StepTxt;
	p_sOpsMagConvLD4StepTxt ACCESS p_OpsMagConvLD4StepTxt;

	p_bOpsTravLifLDInitConv ACCESS p_OpsTravLifLDInitConv;
	p_bOpsTravLifLDAWPosDiff ACCESS p_OpsTravLifLDAWPosDiff;
	p_bOpsTravLifLDExitBrd ACCESS p_OpsTravLifLDExitBrd;
	p_eOpsTravLifPosGo ACCESS p_OpsTravLifLDPosGo;
	p_bOpsTravLifStandby ACCESS p_OpsTravLifStandby;

	p_bOpsLifMagLDUnloading ACCESS p_OpsLifMagLDUnloading;
	p_sOpsLifMagLDStepTxt ACCESS p_OpsLifMagLDStepTxt;

	p_bOpsMagConvLD1InitDone ACCESS p_OpsMagConvLD1InitDone;
	p_bOpsMagConvLD2InitDone ACCESS p_OpsMagConvLD2InitDone;
	p_bOpsMagConvLD3InitDone ACCESS p_OpsMagConvLD3InitDone;
	p_bOpsMagConvLD4InitDone ACCESS p_OpsMagConvLD4InitDone;
	p_bOpsMagConvLD1MagExitedWait ACCESS p_OpsMagConvLD1ExitedWait;
	p_bOpsMagConvLD2MagExitedWait ACCESS p_OpsMagConvLD2ExitedWait;
	p_bOpsMagConvLD3MagExitedWait ACCESS p_OpsMagConvLD3ExitedWait;
	p_bOpsMagConvLD4MagExitedWait ACCESS p_OpsMagConvLD4ExitedWait;
	p_bOpsMagConvLD1NewMagAllw ACCESS p_OpsMagConvLD1NewMagAllw;
	p_bOpsMagConvLD2NewMagAllw ACCESS p_OpsMagConvLD2NewMagAllw;
	p_bOpsMagConvLD3NewMagAllw ACCESS p_OpsMagConvLD3NewMagAllw;
	p_bOpsMagConvLD4NewMagAllw ACCESS p_OpsMagConvLD4NewMagAllw;
	p_bOpsMagConvLD1RlsMagAllw ACCESS p_OpsMagConvLD1RlsMagAllw;
	p_bOpsMagConvLD2RlsMagAllw ACCESS p_OpsMagConvLD2RlsMagAllw;
	p_bOpsMagConvLD3RlsMagAllw ACCESS p_OpsMagConvLD3RlsMagAllw;
	p_bOpsMagConvLD4RlsMagAllw ACCESS p_OpsMagConvLD4RlsMagAllw;
	p_bOpsMagConvLD1RlsMagUmask ACCESS p_OpsMagConvLD1RlsMagUmask;
	p_bOpsMagConvLD2RlsMagUmask ACCESS p_OpsMagConvLD2RlsMagUmask;
	p_bOpsMagConvLD3RlsMagUmask ACCESS p_OpsMagConvLD3RlsMagUmask;
	p_bOpsMagConvLD1ExtMes ACCESS p_OpsMagConvLD1ExtMes;
	p_bOpsMagConvLD2ExtMes ACCESS p_OpsMagConvLD2ExtMes;
	p_bOpsMagConvLD3ExtMes ACCESS p_OpsMagConvLD3ExtMes;
	p_bOpsMagConvLD1HModChgDone ACCESS p_OpsMagConvLD1HModChgDone;
	p_bOpsMagConvLD2HModChgDone ACCESS p_OpsMagConvLD2HModChgDone;
	p_bOpsMagConvLD3HModChgDone ACCESS p_OpsMagConvLD3HModChgDone;

	p_tyDTMagToAGV1 ACCESS p_AGVMag1DTMagToAGV;
	p_tyDTMagToAGV2 ACCESS p_AGVMag2DTMagToAGV;
	p_tyDTMagToAGV3 ACCESS p_AGVMag3DTMagToAGV;
	p_tyDTMagToAGV4 ACCESS p_AGVMag4DTMagToAGV;

	p_tyAGVToDTMag ACCESS p_AGVTagAGVToDTMag;
	p_bAGVOnline ACCESS p_AGVOnline;
	p_bMachineOnline ACCESS p_MachineOnline;
	p_tyDTMagToAGV ACCESS p_DTMagToAGV;
	p_bAGVSimulationOn ACCESS p_AGVSimulationOn;
	p_tyTagToMes ACCESS p_TagToMes;
	p_tyTagFromMes ACCESS p_TagFromMes;

	//Simulation
	p_eSimuStat ACCESS p_SimuStat;
	p_eSimuStatus ACCESS p_SimuStatus;

	p_eSimuSimuStatus ACCESS p_SimuSimuStatus;
	p_bSimuStatusRun ACCESS p_SimuStatusRun;
	p_bSimuStatusStop ACCESS p_SimuStatusStop;
	p_bSimuStatusCycleStop ACCESS p_SimuStatusCycleStop;
	p_bSimuStatusStep ACCESS p_SimuStatusStep;
	p_sNtParamJobNo ACCESS p_NtParamJobNo;
	p_usiNtParamNtAddr ACCESS p_NtParamNtAddr;
	p_eNtParamStat ACCESS p_NtParamStat;
	p_eNtParamStatus ACCESS p_NtParamStatus;
	p_diNtParamLifterAutoSpd ACCESS p_NtParamLifterAutoSpd;
	p_diNtParamTravAutoSpd ACCESS p_NtParamTravAutoSpd;

	//USB Barcode Reader
	p_eUSBRdrStat ACCESS p_USBRdrStat;
	p_eUSBRdrStatus ACCESS p_USBRdrStatus;
	p_sUSBRdrBarcodeOut ACCESS p_USBRdrBarcodeOut;
	p_bUSBDisconnected ACCESS p_USBDisconnected;

	p_eFrmStat ACCESS p_FrmStat;
	p_eFrmStatus ACCESS p_FrmStatus;
	p_sFrmFullMsgRd ACCESS p_FrmFullMsgRd;
	p_sFrmMsgRd	ACCESS p_FrmMsgRd;
	p_bFrmMsgRdValid ACCESS p_FrmMsgRdValid;
	p_uiFrmMsgRdLen ACCESS p_FrmMsgRdLen;

	p_eMtrPshrStat ACCESS p_MtrPshrStat;
	p_eMtrPshrStatus ACCESS p_MtrPshrStatus;
	p_sMtrPshrStatTxt ACCESS p_MtrPshrStatTxt;

	p_eMag1SafetyBarStat ACCESS p_Pneu2SMag1SafetyBarStat;
	p_eMag1SafetyBarStatus ACCESS p_Pneu2SMag1SafetyBarStatus;
	p_sMag1SafetyBarStatTxt ACCESS p_Pneu2SMag1SafetyBarStatTxt;
	p_bMag1SafetyBarExtCtrl ACCESS p_Pneu2SMag1SafetyBarExtCtrl;
	p_bMag1SafetyBarRetCtrl ACCESS p_Pneu2SMag1SafetyBarRetCtrl;
	p_bMag1SafetyBarTwoCtrlOut ACCESS p_Pneu2SMag1SafetyBarTwoCtrlOut;
	p_bMag1SafetyBarExtended ACCESS p_Pneu2SMag1SafetyBarExtended;
	p_bMag1SafetyBarRetracted ACCESS p_Pneu2SMag1SafetyBarRetracted;

	p_eMag2SafetyBarStat ACCESS p_Pneu2SMag2SafetyBarStat;
	p_eMag2SafetyBarStatus ACCESS p_Pneu2SMag2SafetyBarStatus;
	p_sMag2SafetyBarStatTxt ACCESS p_Pneu2SMag2SafetyBarStatTxt;
	p_bMag2SafetyBarExtCtrl ACCESS p_Pneu2SMag2SafetyBarExtCtrl;
	p_bMag2SafetyBarRetCtrl ACCESS p_Pneu2SMag2SafetyBarRetCtrl;
	p_bMag2SafetyBarTwoCtrlOut ACCESS p_Pneu2SMag2SafetyBarTwoCtrlOut;
	p_bMag2SafetyBarExtended ACCESS p_Pneu2SMag2SafetyBarExtended;
	p_bMag2SafetyBarRetracted ACCESS p_Pneu2SMag2SafetyBarRetracted;

	p_eMag3SafetyBarStat ACCESS p_Pneu2SMag3SafetyBarStat;
	p_eMag3SafetyBarStatus ACCESS p_Pneu2SMag3SafetyBarStatus;
	p_sMag3SafetyBarStatTxt ACCESS p_Pneu2SMag3SafetyBarStatTxt;
	p_bMag3SafetyBarExtCtrl ACCESS p_Pneu2SMag3SafetyBarExtCtrl;
	p_bMag3SafetyBarRetCtrl ACCESS p_Pneu2SMag3SafetyBarRetCtrl;
	p_bMag3SafetyBarTwoCtrlOut ACCESS p_Pneu2SMag3SafetyBarTwoCtrlOut;
	p_bMag3SafetyBarExtended ACCESS p_Pneu2SMag3SafetyBarExtended;
	p_bMag3SafetyBarRetracted ACCESS p_Pneu2SMag3SafetyBarRetracted;

	p_diNtParamPullerHeightInMM ACCESS p_NtParamPullerHeightInMM;

	p_eTrolleyLckStat ACCESS p_PneuExtSenTrllyStat;
	p_eTrolleyLckStatus ACCESS p_PneuExtSenTrllyStatus;
	p_sTrolleyLckStatTxt ACCESS p_PneuExtSenTrllyStatTxt;
	p_bTrolleyLckExtCtrl ACCESS p_PneuExtSenTrllyExtCtrl;
	p_bTrolleyLckRetCtrl ACCESS p_PneuExtSenTrllyRetCtrl;
	p_bTrolleyLckTwoCtrlOut ACCESS p_PneuExtSenTrllyTwoCtrlOut;
	p_bTrolleyLckExtended ACCESS p_PneuExtSenTrllyExtended;
	p_bTrolleyLckRetracted ACCESS p_PneuExtSenTrllyRetracted;

	p_eTrolleyLckStat2 ACCESS p_PneuExtSenTrlly2Stat;
	p_eTrolleyLckStatus2 ACCESS p_PneuExtSenTrlly2Status;
	p_sTrolleyLckStatTxt2 ACCESS p_PneuExtSenTrlly2StatTxt;
	p_bTrolleyLckExtCtrl2 ACCESS p_PneuExtSenTrlly2ExtCtrl;
	p_bTrolleyLckRetCtrl2 ACCESS p_PneuExtSenTrlly2RetCtrl;
	p_bTrolleyLckTwoCtrlOut2 ACCESS p_PneuExtSenTrlly2TwoCtrlOut;
	p_bTrolleyLckExtended2 ACCESS p_PneuExtSenTrlly2Extended;
	p_bTrolleyLckRetracted2 ACCESS p_PneuExtSenTrlly2Retracted;

	p_ePPStat ACCESS p_PPStat;
	p_ePPStatus ACCESS p_PPStatus;
	p_sPPStatTxt ACCESS p_PPStatTxt;
	p_bPPPwrOn ACCESS p_PPPwrOn;
	p_bPPIsHomed ACCESS p_PPIsHomed;
	p_bPPPosDiff ACCESS p_PPPosDiff;
	p_bPPAxisErr ACCESS p_PPAxisErr;
	p_udiPPAxisErrID ACCESS p_PPAxisErrID;
	p_sPPAxisErrTxt ACCESS p_PPAxisErrTxt;
	p_bPPFwdLmtSen ACCESS p_PPFwdLmtSen;
	p_bPPRevLmtSen ACCESS p_PPRevLmtSen;
	p_diPPActualPos ACCESS p_PPActualPos;
	p_bPPJogging ACCESS p_PPJogging;
	p_bPPExtSen ACCESS p_PPExtSen;
	p_bPPRetSen ACCESS p_DIPullerRetRS;

	p_tyMcAlmData ACCESS p_McAlmData;

	//new for Hermes 1.3
	p_bRmtUpdateUIData ACCESS p_RmtHermesUpdateUIData;//new for Hermes 1.3
	p_bSvyUpdateUIData ACCESS p_SvyHermesUpdateUIData;//new for Hermes 1.3
	p_bRcvBoardInfoOk ACCESS p_SvyHermesUpdateUIData;//p_USHermesRcvBoardInfoOk;//new for Hermes 1.3
	p_bRcvBoardInfoIncompl ACCESS p_SvyHermesUpdateUIData;//p_USHermesRcvbBoardInfoIncompl;//new for Hermes 1.3
	p_bTransportFinished ACCESS p_DSHermesATransportFinishedSnd;//new for Hermes 1.3
	p_sWorkOrderId ACCESS p_SvyHermesWorkOrderId; //Work Order Id from SupervisoryHermes
	p_bWaitDecision ACCESS p_StartupWaitDecision;//new for Hermes 1.3

	p_tySendWorkOrderData ACCESS p_SvyHermesSendWorkOrderData;
	p_tySvyHermesSendWorkOrderData ACCESS p_SvyHermesSendWorkOrderData;
	p_tySvyHermesBypassSendWOData ACCESS p_SvyHermesBypassSendWOData;
//	p_bOpsConvWaitForTopUpBrd ACCESS p_OpsConvWaitForTopUpBrd;
	p_diReqLoaderWidthInUM ACCESS p_ReqLoaderWidthInUM;
	p_bQueryBypassWorkOrder ACCESS p_QueryBypassWorkOrder;
	p_bReplyBypassWorkOrderInfo ACCESS p_ReplyBypassWorkOrderInfo;
	p_bRcvWorkOrderInfo1 ACCESS p_RcvWorkOrderInfo1;
//	p_bOpsPneuStepLifToLoadPos ACCESS p_OpsPneuStepLifToLoadPos;
	p_bNewIncomingBoard ACCESS p_NewIncomingBoard;

	//AutoRcp
	p_diLinkAutoRcpMag1Pitch ACCESS p_diAutoRcpMag1Pitch;
	p_diLinkAutoRcpMag1MinSlt ACCESS p_diAutoRcpMag1MinSlt;
	p_diLinkAutoRcpMag1MaxSlt ACCESS p_diAutoRcpMag1MaxSlt;

	p_diLinkAutoRcpMag2Pitch ACCESS p_diAutoRcpMag2Pitch;
	p_diLinkAutoRcpMag2MinSlt ACCESS p_diAutoRcpMag2MinSlt;
	p_diLinkAutoRcpMag2MaxSlt ACCESS p_diAutoRcpMag2MaxSlt;

	p_diLinkAutoRcpMag3Pitch ACCESS p_diAutoRcpMag3Pitch;
	p_diLinkAutoRcpMag3MinSlt ACCESS p_diAutoRcpMag3MinSlt;
	p_diLinkAutoRcpMag3MaxSlt ACCESS p_diAutoRcpMag3MaxSlt;
	p_ausiSvyMagAccOrder ACCESS p_SvyHermesMagAccOrder;
	p_tyAutoRcpMagRcp ACCESS p_AutoRcpMagRcp;//display in prod name

END_ACTION
```

#### Act_InitLocal.st - Do Not Change!!!
```iecst
(** 2019-03-25 **)
ACTION Act_InitLocal:

	//Input Reference Link To Local Variable
	p_eAct ACCESS ADR(eAct);

	p_sUSBRdrBarcodeOut ACCESS ADR(sUSBBarcode);
	p_bUSBDisconnected ACCESS ADR(bUSBDisconnected);
END_ACTION
```

#### Act_Initial.st - Change By Project
```iecst
(** 2019-01-03 **)
ACTION Act_Initial:

	//Initial
	sStatTxt	:= a_sStatText[eStat];

	//for simulation
	fbSDOWriteAccT.pDevice := ADR(sDevice);
	fbSDOWriteAccT.node	 := 18;//Trav dec.

//	fbSDOWriteAccT.index	:= 16#6083;
//	fbSDOWriteAccT.subindex	:= 0;
//	fbSDOWriteAccT.datalen	:= 4;

	fbSDOWriteAccL.pDevice := ADR(sDevice);
	fbSDOWriteAccL.node	 := 17;//Lifter

//	fbSDOWriteAccL.index	:= 16#6083;
//	fbSDOWriteAccL.subindex	:= 0;
//	fbSDOWriteAccL.datalen	:= 4;
END_ACTION
```

#### Act_Main.st - Do Not Change!!!
```iecst
(** 2019-03-25 **)
ACTION Act_Main:

	//Main
	CASE eStat OF

		UIActIdle:
			IF eStatus <> Idle THEN	//Reset Data
				//Private

				sStatTxt	:= a_sStatText[eStat];

				eUIInit	:= UIInitialC0005;

			END_IF

			eStatus	:= Idle;

		UIActInitial:
			IF eStatus = Idle OR eStatus = Busy THEN

				eStatus	:= Busy;

				sStatTxt	:= a_sStatText[eStat];

				CASE eUIInit OF
					UIInitialC0005:
						Act_Main_C0005;
						eUIInit	:= UIInitialC0007;

					UIInitialC0007:
						Act_Main_C0007;
						eUIInit	:= UIInitialP0000;

					UIInitialP0000:
						Act_Main_P0000;
						eUIInit	:= UIInitialP0002;

					UIInitialP0002:
						Act_Main_P0002;
						eUIInit	:= UIInitialP0200;

					UIInitialP0200:
						Act_Main_P0200;
						eUIInit	:= UIInitialP0201;

					UIInitialP0201:
						Act_Main_P0201;
						eUIInit	:= UIInitialP0202;

					UIInitialP0202:
						Act_Main_P0202;
						eUIInit	:= UIInitialP0203;

					UIInitialP0203:
						Act_Main_P0203;
						eUIInit	:= UIInitialP0204;

					UIInitialP0204:
						Act_Main_P0204;
						eUIInit	:= UIInitialP0205;

					UIInitialP0205:
						Act_Main_P0205;
						eUIInit	:= UIInitialP0206;

					UIInitialP0206:
						Act_Main_P0206;
						eUIInit	:= UIInitialP0300;

					UIInitialP0300:
						Act_Main_P0300;
						eUIInit	:= UIInitialP0400;

					UIInitialP0400:
						Act_Main_P0400;
						eUIInit	:= UIInitialP0410;

					UIInitialP0410:
						Act_Main_P0410;
						eUIInit	:= UIInitialP0800;

					UIInitialP0800:
						Act_Main_P0800;
						eUIInit	:= UIInitialP0900;

					UIInitialP0900:
						Act_Main_P0900;
						eUIInit	:= UIInitialP0910;

					UIInitialP0910:
						Act_Main_P0910;
						eUIInit	:= UIInitialP0920;

					UIInitialP0920:
						Act_Main_P0920;
						eUIInit	:= UIInitialP0921;

					UIInitialP0921:
						Act_Main_P0921;
						eUIInit	:= UIInitialP0923;

					UIInitialP0923:
						Act_Main_P0923;
						eUIInit	:= UIInitialP0930;

					UIInitialP0930:
						Act_Main_P0930;
						eUIInit	:= UIInitialP0931;

					UIInitialP0931:
						Act_Main_P0931;
						eUIInit	:= UIInitialP0932;

					UIInitialP0932:
						Act_Main_P0932;
						eUIInit	:= UIInitialP0933;

					UIInitialP0933:
						Act_Main_P0933;
						eUIInit	:= UIInitialP0934;

					UIInitialP0934:
						Act_Main_P0934;
						eUIInit	:= UIInitialP0935;

					UIInitialP0935:
						Act_Main_P0935;
						eUIInit	:= UIInitialP0936;

					UIInitialP0936:
						Act_Main_P0936;
						eUIInit	:= UIInitialP0937;

					UIInitialP0937:
						Act_Main_P0937;
						eUIInit	:= UIInitialP0939;

					UIInitialP0939:
						Act_Main_P0939;
						eUIInit	:= UIInitialP0940;

					UIInitialP0940:
						Act_Main_P0940;
						eUIInit	:= UIInitialP0950;

					UIInitialP0950:
						Act_Main_P0950;
						eUIInit	:= UIInitialP1000;

					UIInitialP1000:
						Act_Main_P1000;
						eUIInit	:= UIInitialP1020;

					UIInitialP1020:
						Act_Main_P1020;
						eUIInit	:= UIInitialP1021;

					UIInitialP1021:
						Act_Main_P1021;
						eUIInit	:= UIInitialP1022;

					UIInitialP1022:
						Act_Main_P1022;
						eUIInit	:= UIInitialP1023;

					UIInitialP1023:
						Act_Main_P1023;
						eUIInit	:= UIInitialP1024;

					UIInitialP1024:
						Act_Main_P1024;
						eUIInit	:= UIInitialP1025;

					UIInitialP1025:
						Act_Main_P1025;
						eUIInit	:= UIInitialP1026;

					UIInitialP1026:
						Act_Main_P1026;
						eUIInit	:= UIInitialP1027;

					UIInitialP1027:
						Act_Main_P1027;
						eUIInit	:= UIInitialP1028;

					UIInitialP1028:
						Act_Main_P1028;
						eUIInit	:= UIInitialP1030;

					UIInitialP1030:
						Act_Main_P1030;
						eUIInit	:= UIInitialP1031;

					UIInitialP1031:
						Act_Main_P1031;
						eUIInit	:= UIInitialP1040;

					UIInitialP1040:
						Act_Main_P1040;
						eUIInit	:= UIInitialP1050;

					UIInitialP1050:
						Act_Main_P1050;
						eUIInit	:= UIInitialP1080;

					UIInitialP1080:
						Act_Main_P1080;
						eUIInit	:= UIInitialP1081;

					UIInitialP1081:
						Act_Main_P1081;
						eUIInit	:= UIInitialDone;

					UIInitialDone:
						tyMcParamWr					:= p_tyMcParamCurr;

						tyProdRcpCurrRcpWr			:= p_tyProdRcpCurrRcp0;

						tyMagRcpCurrRcpWr			:= p_tyMagRcpCurrRcp;

						tyUsrMgmtAccessRightLvl1Wr	:= p_tyUsrMgmtFullData.tyAccessRightLvl1;
						tyUsrMgmtAccessRightLvl2Wr	:= p_tyUsrMgmtFullData.tyAccessRightLvl2;
						tyUsrMgmtAccessRightLvl3Wr	:= p_tyUsrMgmtFullData.tyAccessRightLvl3;

						a_tyHermesDSParamWr			:= p_tyHermesConfiguration.a_tyDSParam;

						eStatus	:= Done;

				END_CASE

			END_IF

	END_CASE

END_ACTION
```

#### Package Logical/UI/UI/Act_Main - Change By Project

#### Act_Main_C0005.st
```iecst
(** 2018-12-21 **)
ACTION Act_Main_C0005:

	tyCommon.tyMain.tyBtnBuzzer.uiRtStat.0	:= p_tyNtParamCurr.tyDOSettings.diBuzzer = 0;

	fUIInRtStatHide(ADR(tyCommon.tyMain.tyBtnAlarm.uiRtStat));

END_ACTION
```

#### Act_Main_P0000.st
```iecst
ACTION Act_Main_P0000:

	tyProperty.tyVisu.uiSSaverTm	:= p_tyMcParamCurr.uiSSaverTmInSec;

END_ACTION
```

#### Act_Main_P0200.st
```iecst
(** 2018-12-21 **)
ACTION Act_Main_P0200:

	//Display
	tyP0200OpsGen.tyOps.tyTxtMag3Slt.uiRtStat.0		:= NOT(p_tyNtParamCurr.eProjMag = LDMagTriple OR p_tyNtParamCurr.eProjMag = LDMagQuadruple);
	tyP0200OpsGen.tyOps.tyTxtBackslash3.uiRtStat.0	:= NOT(p_tyNtParamCurr.eProjMag = LDMagTriple OR p_tyNtParamCurr.eProjMag = LDMagQuadruple);
	tyP0200OpsGen.tyOps.tyNumMag3AvlQty.uiRtStat.0	:= NOT(p_tyNtParamCurr.eProjMag = LDMagTriple OR p_tyNtParamCurr.eProjMag = LDMagQuadruple);
	tyP0200OpsGen.tyOps.tyNumMag3TtlSlt.uiRtStat.0	:= NOT(p_tyNtParamCurr.eProjMag = LDMagTriple OR p_tyNtParamCurr.eProjMag = LDMagQuadruple);

	//L to R
	tyP0200OpsGen.tyOps.tyHotspotOps2Mag1.uiRtStat.0	:= NOT(p_tyNtParamCurr.eProjMag = LDMagDual) OR p_tyNtParamCurr.bUIConvDirRL = TRUE;
	tyP0200OpsGen.tyOps.tyHotspotOps2Mag2.uiRtStat.0	:= NOT(p_tyNtParamCurr.eProjMag = LDMagDual) OR p_tyNtParamCurr.bUIConvDirRL = TRUE;
	tyP0200OpsGen.tyOps.tyHotspotOps3Mag1.uiRtStat.0	:= NOT(p_tyNtParamCurr.eProjMag = LDMagTriple) OR p_tyNtParamCurr.bUIConvDirRL = TRUE;
	tyP0200OpsGen.tyOps.tyHotspotOps3Mag2.uiRtStat.0	:= NOT(p_tyNtParamCurr.eProjMag = LDMagTriple) OR p_tyNtParamCurr.bUIConvDirRL = TRUE;
	tyP0200OpsGen.tyOps.tyHotspotOps3Mag3.uiRtStat.0	:= NOT(p_tyNtParamCurr.eProjMag = LDMagTriple) OR p_tyNtParamCurr.bUIConvDirRL = TRUE;
	tyP0200OpsGen.tyOps.tyHotspotOpsTravLifter.uiRtStat.0		:= p_tyNtParamCurr.bUIConvDirRL = TRUE;

	tyP0200OpsGen.tyOps.tyHotspotOps4Mag1.uiRtStat.0	:= NOT(p_tyNtParamCurr.eProjMag = LDMagQuadruple) OR p_tyNtParamCurr.bUIConvDirRL = TRUE;
	tyP0200OpsGen.tyOps.tyHotspotOps4Mag2.uiRtStat.0	:= NOT(p_tyNtParamCurr.eProjMag = LDMagQuadruple) OR p_tyNtParamCurr.bUIConvDirRL = TRUE;
	tyP0200OpsGen.tyOps.tyHotspotOps4Mag3.uiRtStat.0	:= NOT(p_tyNtParamCurr.eProjMag = LDMagQuadruple) OR p_tyNtParamCurr.bUIConvDirRL = TRUE;
	tyP0200OpsGen.tyOps.tyHotspotOps4Mag4.uiRtStat.0	:= NOT(p_tyNtParamCurr.eProjMag = LDMagQuadruple) OR p_tyNtParamCurr.bUIConvDirRL = TRUE;

	//R to L
	tyP0200OpsGen.tyOps.tyHotspotOps2Mag1RToL.uiRtStat.0	:= NOT(p_tyNtParamCurr.eProjMag = LDMagDual) OR p_tyNtParamCurr.bUIConvDirRL = FALSE;
	tyP0200OpsGen.tyOps.tyHotspotOps2Mag2RToL.uiRtStat.0	:= NOT(p_tyNtParamCurr.eProjMag = LDMagDual)OR p_tyNtParamCurr.bUIConvDirRL = FALSE;
//	tyP0200OpsGen.tyOps.tyHotspotOps3Mag1RToL.uiRtStat.0	:= NOT(p_tyNtParamCurr.eProjMag = LDMagTriple)OR p_tyNtParamCurr.bUIConvDirRL = FALSE;
//	tyP0200OpsGen.tyOps.tyHotspotOps3Mag2RToL.uiRtStat.0	:= NOT(p_tyNtParamCurr.eProjMag = LDMagTriple)OR p_tyNtParamCurr.bUIConvDirRL = FALSE;
//	tyP0200OpsGen.tyOps.tyHotspotOps3Mag3RToL.uiRtStat.0	:= NOT(p_tyNtParamCurr.eProjMag = LDMagTriple)OR p_tyNtParamCurr.bUIConvDirRL = FALSE;
	tyP0200OpsGen.tyOps.tyHotspotOpsTravLifterRToL.uiRtStat.0		:= p_tyNtParamCurr.bUIConvDirRL = FALSE;

	//Machine Bitmap //mc.default 31
	IF p_tyNtParamCurr.eProjMag = LDMagDual AND p_tyNtParamCurr.bMagAutoVerifyPrep = TRUE THEN
		tyP0200OpsGen.tyOps.tyBitmapMc.uiValueIdx	:= 200;
	ELSIF p_tyNtParamCurr.eProjMag = LDMagDual AND p_tyNtParamCurr.sJobNo = '2023-0258A01' THEN //AT&S (RL)
		tyP0200OpsGen.tyOps.tyBitmapMc.uiValueIdx	:= 440-31;
	ELSIF p_tyNtParamCurr.eProjMag = LDMagDual AND p_tyNtParamCurr.sJobNo = '2023-0276A01' THEN //clarion (RL)
		tyP0200OpsGen.tyOps.tyBitmapMc.uiValueIdx	:= 470-31;
	ELSIF p_tyNtParamCurr.eProjMag = LDMagTriple AND p_tyNtParamCurr.bProjLifterMagPlatform THEN
		tyP0200OpsGen.tyOps.tyBitmapMc.uiValueIdx	:= 400;
	ELSIF p_tyNtParamCurr.eProjMag = LDMagTriple AND p_tyNtParamCurr.bProjLifterMagPlatform = FALSE AND p_tyNtParamCurr.bProjCurtainSenPrep THEN
		tyP0200OpsGen.tyOps.tyBitmapMc.uiValueIdx	:= 360-31;
	ELSIF p_tyNtParamCurr.eProjMag = LDMagTriple THEN
		tyP0200OpsGen.tyOps.tyBitmapMc.uiValueIdx	:= 214;
	ELSIF p_tyNtParamCurr.eProjMag = LDMagQuadruple THEN
		tyP0200OpsGen.tyOps.tyBitmapMc.uiValueIdx	:= 51;
	ELSE
		tyP0200OpsGen.tyOps.tyBitmapMc.uiValueIdx	:= 0;
	END_IF

	//Communication
	tyP0200OpsGen.tyDSCommB.tyLyr.uiRtStat.0 := NOT(p_tyNtParamCurr.bProjLaneBPrep);

	//Direction
	CASE p_tyNtParamCurr.eProjConvDir OF
		ConvDirLToR:
			tyP0200OpsGen.tyOps.tyBitmapDir1.usiValueIdx	:= 0;	// -->>
			tyP0200OpsGen.tyOps.tyBitmapDir2.usiValueIdx	:= 0;	// -->>
		ConvDirRToL:
			tyP0200OpsGen.tyOps.tyBitmapDir1.usiValueIdx	:= 1;	// <<--
			tyP0200OpsGen.tyOps.tyBitmapDir2.usiValueIdx	:= 1;	// <<--
	END_CASE
	IF p_tyNtParamCurr.bUIConvDirRL THEN
		tyP0200OpsGen.tyOps.tyBitmapDir1.usiValueIdx	:= 1;	// <<--
		tyP0200OpsGen.tyOps.tyBitmapDir2.usiValueIdx	:= 1;	// <<--
	ELSE
		tyP0200OpsGen.tyOps.tyBitmapDir1.usiValueIdx	:= 0;	// -->>
		tyP0200OpsGen.tyOps.tyBitmapDir2.usiValueIdx	:= 0;	// -->>
	END_IF

	//Hide Warning Bitmap for LF
	fUIInRtStatHide(ADR(tyP0200OpsGen.tyOps.tyTxtLdrInActiveCtrl.uiRtStat));
	fUIInRtStatHide(ADR(tyP0201OpsTravLifter.tyOps.tyTxtLdrInActiveCtrl.uiRtStat));
	fUIInRtStatHide(ADR(tyP0202OpsMag1.tyOps.tyTxtLdrInActiveCtrl.uiRtStat));
	fUIInRtStatHide(ADR(tyP0203OpsMag2.tyOps.tyTxtLdrInActiveCtrl.uiRtStat));
	fUIInRtStatHide(ADR(tyP0204OpsMag3.tyOps.tyTxtLdrInActiveCtrl.uiRtStat));
	fUIInRtStatHide(ADR(tyP0206OpsMag4.tyOps.tyTxtLdrInActiveCtrl.uiRtStat));

	fUIInRtStatHide(ADR(tyP0200OpsGen.tyOps.tyBitmapWarningLF.uiRtStat));
	fUIInRtStatHide(ADR(tyP0201OpsTravLifter.tyOps.tyBitmapWarningLF.uiRtStat));
	fUIInRtStatHide(ADR(tyP0202OpsMag1.tyOps.tyBitmapWarningLF.uiRtStat));
	fUIInRtStatHide(ADR(tyP0203OpsMag2.tyOps.tyBitmapWarningLF.uiRtStat));
	fUIInRtStatHide(ADR(tyP0204OpsMag3.tyOps.tyBitmapWarningLF.uiRtStat));
	fUIInRtStatHide(ADR(tyP0206OpsMag4.tyOps.tyBitmapWarningLF.uiRtStat));

	IF p_tyNtParamCurr.eProjMag <> LDMagQuadruple THEN
		fUIInRtStatHide(ADR(tyP0200OpsGen.tyOps.tyTxtMag4Slt.uiRtStat));
		fUIInRtStatHide(ADR(tyP0200OpsGen.tyOps.tyNumMag4AvlQty.uiRtStat));
		fUIInRtStatHide(ADR(tyP0200OpsGen.tyOps.tyNumMag4TtlSlt.uiRtStat));

		fUIInRtStatHide(ADR(tyP0200OpsGen.tyOps.tyNumMaxSltRangeRear.uiRtStat));
		fUIInRtStatHide(ADR(tyP0200OpsGen.tyOps.tyNumMinSltRangeRear.uiRtStat));

		fUIInRtStatHide(ADR(tyP0200OpsGen.tyOps.tyNumPitchRear.uiRtStat));

	END_IF

	tyP0200OpsGen.tyOps.tyBtnBarCodeScan.uiRtStat.0 := NOT ((p_tyNtParamCurr.bUSBScannerPrep OR p_tyNtParamCurr.bRS232ScannerPrep) AND p_tyMcParamCurr.bScannerEn);
	tyP0200OpsGen.tyOps.tyBitmapBarCodeScan.uiRtStat.0 := NOT ((p_tyNtParamCurr.bUSBScannerPrep OR p_tyNtParamCurr.bRS232ScannerPrep) AND p_tyMcParamCurr.bScannerEn);
	tyP0200OpsGen.tyBarCodeScan.tyStringBarCode.sValue  := '';
	tyP0200OpsGen.tyBarCodeScan.tyStringWorkOrder.sValue  := '';

	tyP0200OpsGen.tyOps.tyHotspotOpsAIV.uiRtStat.0 := NOT (p_tyNtParamCurr.bProjAGVPrep);

	//Trolley unlck btn
	tyP0200OpsGen.tyOps.tyBtnTrolleyUnlck1.uiRtStat := NOT(p_tyNtParamCurr.bProjTrolleyLckPrep);
	tyP0200OpsGen.tyOps.tyBtnTrolleyUnlck2.uiRtStat := NOT(p_tyNtParamCurr.bProjTrolleyLckPrep);

END_ACTION
```
